// Mitsubishi GX Developer project: 12-202_20140305   PLC: FX3U

PROGRAM MAIN
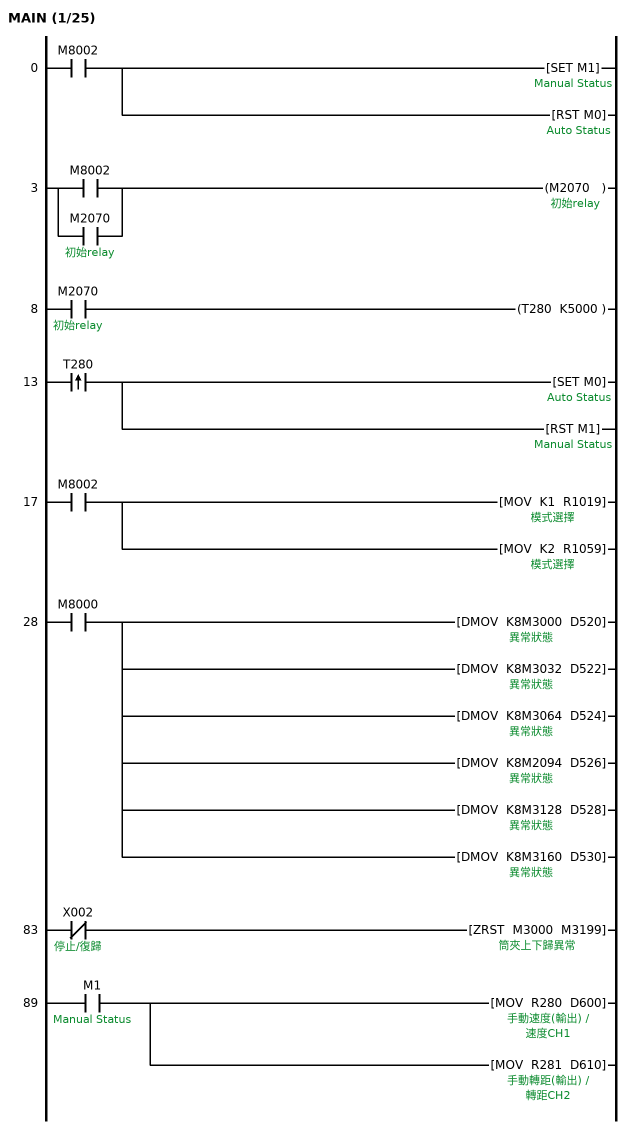
0     LD      M8002
      SET     M1  ; Manual Status
      RST     M0  ; Auto Status
3     LD      M8002
      OR      M2070  ; 初始relay
      OUT     M2070  ; 初始relay
8     LD      M2070  ; 初始relay
      OUT     T280 K5000
13    LDP     T280
      SET     M0  ; Auto Status
      RST     M1  ; Manual Status
17    LD      M8002
      MOV     K1 R1019  ; 模式選擇
      MOV     K2 R1059  ; 模式選擇
28    LD      M8000
      DMOV    K8M3000 D520  ; 筒夾上下歸異常 / 異常狀態
      DMOV    K8M3032 D522  ; 異常狀態
      DMOV    K8M3064 D524  ; 異常狀態
      DMOV    K8M2094 D526  ; 異常狀態
      DMOV    K8M3128 D528  ; 異常狀態
      DMOV    K8M3160 D530  ; 異常狀態
83    LDI     X002  ; 停止/復歸
      ZRST    M3000 M3199
89    LD      M1  ; Manual Status
      MOV     R280 D600  ; 手動速度(輸出) / 速度CH1
      MOV     R281 D610  ; 手動轉距(輸出) / 轉距CH2
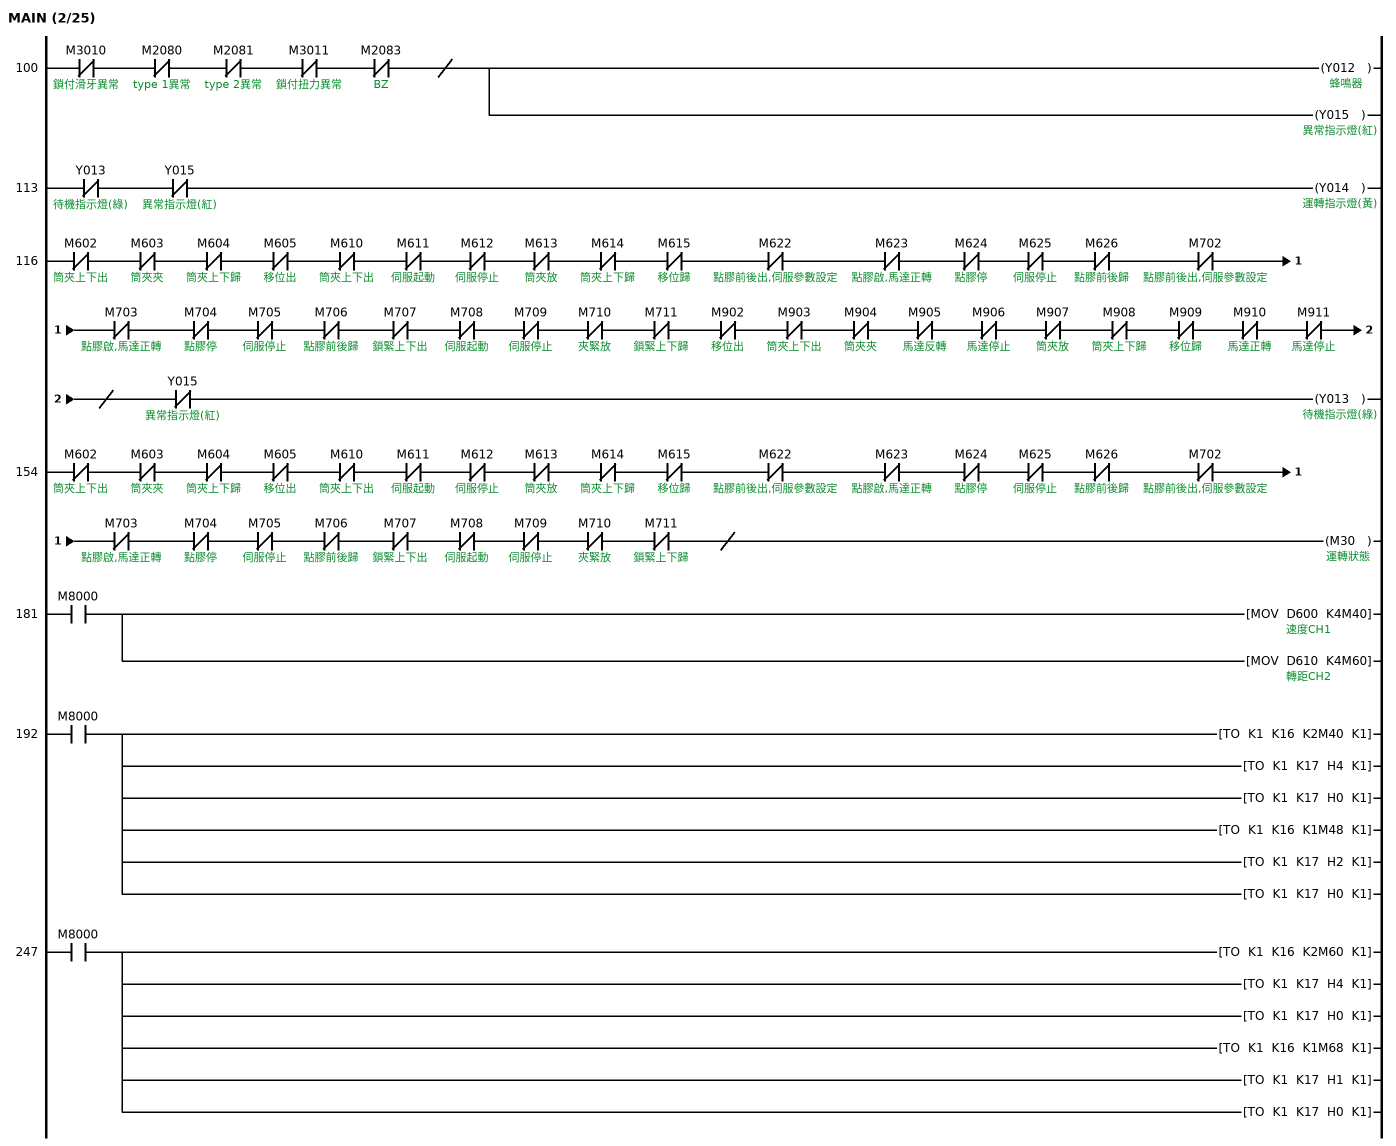
100   LDI     M3010  ; 鎖付滑牙異常
      ANI     M2080  ; type 1異常
      ANI     M2081  ; type 2異常
      ANI     M3011  ; 鎖付扭力異常
      ANI     M2083  ; BZ
      INV
      OUT     Y012  ; 蜂鳴器
      OUT     Y015  ; 異常指示燈(紅)
113   LDI     Y013  ; 待機指示燈(綠)
      ANI     Y015  ; 異常指示燈(紅)
      OUT     Y014  ; 運轉指示燈(黃)
116   LDI     M602  ; 筒夾上下出
      ANI     M603  ; 筒夾夾
      ANI     M604  ; 筒夾上下歸
      ANI     M605  ; 移位出
      ANI     M610  ; 筒夾上下出
      ANI     M611  ; 伺服起動
      ANI     M612  ; 伺服停止
      ANI     M613  ; 筒夾放
      ANI     M614  ; 筒夾上下歸
      ANI     M615  ; 移位歸
      ANI     M622  ; 點膠前後出,伺服參數設定
      ANI     M623  ; 點膠啟,馬達正轉
      ANI     M624  ; 點膠停
      ANI     M625  ; 伺服停止
      ANI     M626  ; 點膠前後歸
      ANI     M702  ; 點膠前後出,伺服參數設定
      ANI     M703  ; 點膠啟,馬達正轉
      ANI     M704  ; 點膠停
      ANI     M705  ; 伺服停止
      ANI     M706  ; 點膠前後歸
      ANI     M707  ; 鎖緊上下出
      ANI     M708  ; 伺服起動
      ANI     M709  ; 伺服停止
      ANI     M710  ; 夾緊放
      ANI     M711  ; 鎖緊上下歸
      ANI     M902  ; 移位出
      ANI     M903  ; 筒夾上下出
      ANI     M904  ; 筒夾夾
      ANI     M905  ; 馬達反轉
      ANI     M906  ; 馬達停止
      ANI     M907  ; 筒夾放
      ANI     M908  ; 筒夾上下歸
      ANI     M909  ; 移位歸
      ANI     M910  ; 馬達正轉
      ANI     M911  ; 馬達停止
      INV
      ANI     Y015  ; 異常指示燈(紅)
      OUT     Y013  ; 待機指示燈(綠)
154   LDI     M602  ; 筒夾上下出
      ANI     M603  ; 筒夾夾
      ANI     M604  ; 筒夾上下歸
      ANI     M605  ; 移位出
      ANI     M610  ; 筒夾上下出
      ANI     M611  ; 伺服起動
      ANI     M612  ; 伺服停止
      ANI     M613  ; 筒夾放
      ANI     M614  ; 筒夾上下歸
      ANI     M615  ; 移位歸
      ANI     M622  ; 點膠前後出,伺服參數設定
      ANI     M623  ; 點膠啟,馬達正轉
      ANI     M624  ; 點膠停
      ANI     M625  ; 伺服停止
      ANI     M626  ; 點膠前後歸
      ANI     M702  ; 點膠前後出,伺服參數設定
      ANI     M703  ; 點膠啟,馬達正轉
      ANI     M704  ; 點膠停
      ANI     M705  ; 伺服停止
      ANI     M706  ; 點膠前後歸
      ANI     M707  ; 鎖緊上下出
      ANI     M708  ; 伺服起動
      ANI     M709  ; 伺服停止
      ANI     M710  ; 夾緊放
      ANI     M711  ; 鎖緊上下歸
      INV
      OUT     M30  ; 運轉狀態
181   LD      M8000
      MOV     D600 K4M40  ; DA用
      MOV     D610 K4M60  ; DA用
192   LD      M8000
      TO      K1 K16 K2M40 K1
      TO      K1 K17 H4 K1
      TO      K1 K17 H0 K1
      TO      K1 K16 K1M48 K1  ; DA用
      TO      K1 K17 H2 K1
      TO      K1 K17 H0 K1
247   LD      M8000
      TO      K1 K16 K2M60 K1
      TO      K1 K17 H4 K1
      TO      K1 K17 H0 K1
      TO      K1 K16 K1M68 K1  ; DA用
      TO      K1 K17 H1 K1
      TO      K1 K17 H0 K1
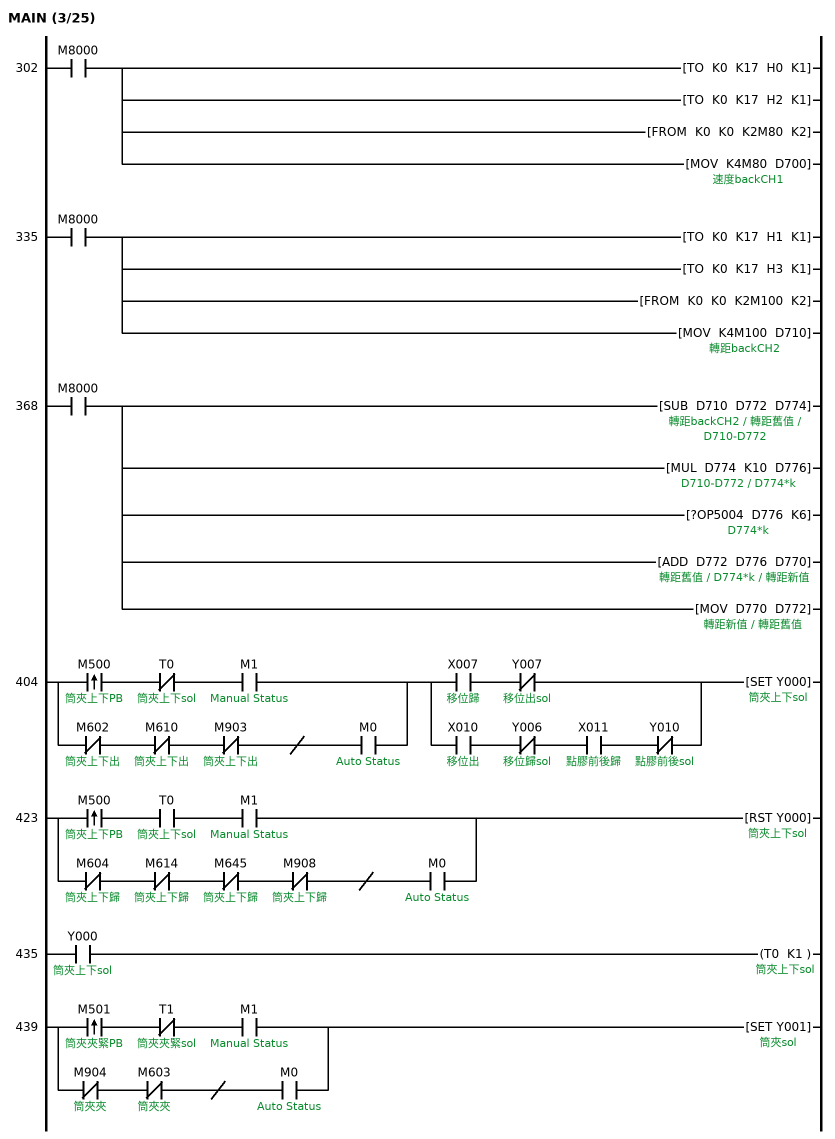
302   LD      M8000
      TO      K0 K17 H0 K1
      TO      K0 K17 H2 K1
      FROM    K0 K0 K2M80 K2  ; AD用
      MOV     K4M80 D700  ; 速度backCH1
335   LD      M8000
      TO      K0 K17 H1 K1
      TO      K0 K17 H3 K1
      FROM    K0 K0 K2M100 K2  ; AD用
      MOV     K4M100 D710  ; 轉距backCH2
368   LD      M8000
      SUB     D710 D772 D774  ; 轉距舊值 / D710-D772
      MUL     D774 K10 D776  ; D774*k
      ?OP5004 D776 K6
      ADD     D772 D776 D770  ; 轉距新值
      MOV     D770 D772
404   LDP     M500  ; 筒夾上下PB
      ANI     T0  ; 筒夾上下sol
      AND     M1  ; Manual Status
      LDI     M602  ; 筒夾上下出
      ANI     M610  ; 筒夾上下出
      ANI     M903  ; 筒夾上下出
      INV
      AND     M0  ; Auto Status
      ORB
      LD      X007  ; 移位歸
      ANI     Y007  ; 移位出sol
      LD      X010  ; 移位出
      ANI     Y006  ; 移位歸sol
      AND     X011  ; 點膠前後歸
      ANI     Y010  ; 點膠前後sol
      ORB
      ANB
      SET     Y000  ; 筒夾上下sol
423   LDP     M500  ; 筒夾上下PB
      AND     T0  ; 筒夾上下sol
      AND     M1  ; Manual Status
      LDI     M604  ; 筒夾上下歸
      ANI     M614  ; 筒夾上下歸
      ANI     M645  ; 筒夾上下歸
      ANI     M908  ; 筒夾上下歸
      INV
      AND     M0  ; Auto Status
      ORB
      RST     Y000  ; 筒夾上下sol
435   LD      Y000  ; 筒夾上下sol
      OUT     T0 K1  ; 筒夾上下sol
439   LDP     M501  ; 筒夾夾緊PB
      ANI     T1  ; 筒夾夾緊sol
      AND     M1  ; Manual Status
      LDI     M904  ; 筒夾夾
      ANI     M603  ; 筒夾夾
      INV
      AND     M0  ; Auto Status
      ORB
      SET     Y001  ; 筒夾sol
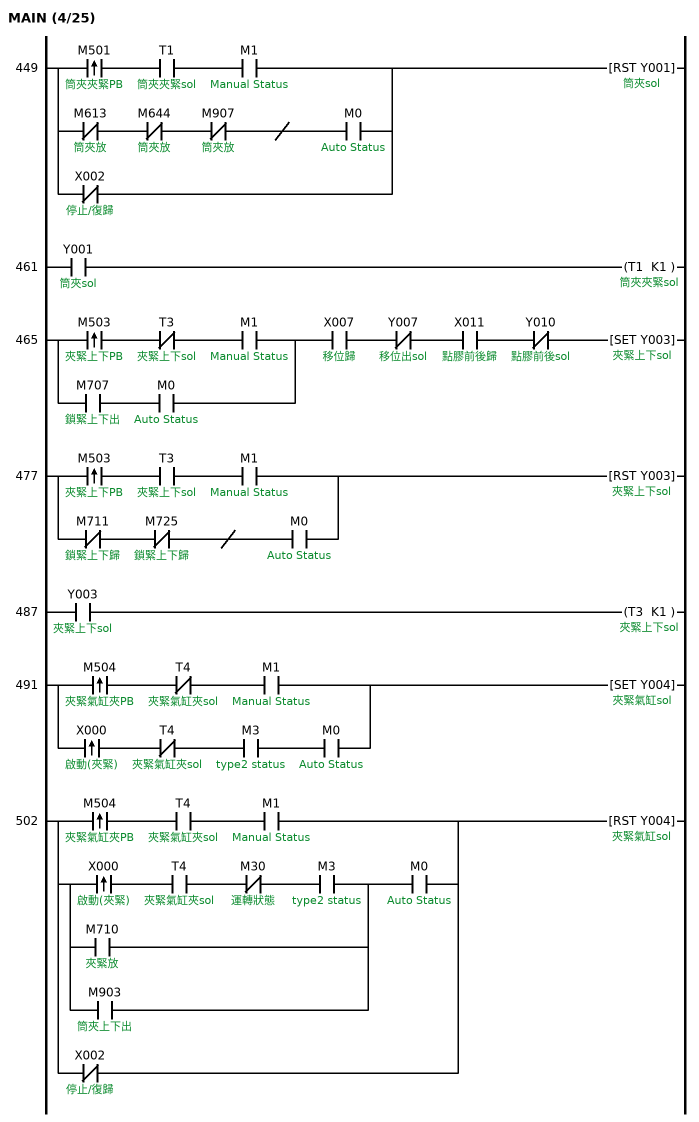
449   LDP     M501  ; 筒夾夾緊PB
      AND     T1  ; 筒夾夾緊sol
      AND     M1  ; Manual Status
      LDI     M613  ; 筒夾放
      ANI     M644  ; 筒夾放
      ANI     M907  ; 筒夾放
      INV
      AND     M0  ; Auto Status
      ORB
      ORI     X002  ; 停止/復歸
      RST     Y001  ; 筒夾sol
461   LD      Y001  ; 筒夾sol
      OUT     T1 K1  ; 筒夾夾緊sol
465   LDP     M503  ; 夾緊上下PB
      ANI     T3  ; 夾緊上下sol
      AND     M1  ; Manual Status
      LD      M707  ; 鎖緊上下出
      AND     M0  ; Auto Status
      ORB
      AND     X007  ; 移位歸
      ANI     Y007  ; 移位出sol
      AND     X011  ; 點膠前後歸
      ANI     Y010  ; 點膠前後sol
      SET     Y003  ; 夾緊上下sol
477   LDP     M503  ; 夾緊上下PB
      AND     T3  ; 夾緊上下sol
      AND     M1  ; Manual Status
      LDI     M711  ; 鎖緊上下歸
      ANI     M725  ; 鎖緊上下歸
      INV
      AND     M0  ; Auto Status
      ORB
      RST     Y003  ; 夾緊上下sol
487   LD      Y003  ; 夾緊上下sol
      OUT     T3 K1  ; 夾緊上下sol
491   LDP     M504  ; 夾緊氣缸夾PB
      ANI     T4  ; 夾緊氣缸夾sol
      AND     M1  ; Manual Status
      LDP     X000  ; 啟動(夾緊)
      ANI     T4  ; 夾緊氣缸夾sol
      AND     M3  ; type2 status
      AND     M0  ; Auto Status
      ORB
      SET     Y004  ; 夾緊氣缸sol
502   LDP     M504  ; 夾緊氣缸夾PB
      AND     T4  ; 夾緊氣缸夾sol
      AND     M1  ; Manual Status
      LDP     X000  ; 啟動(夾緊)
      AND     T4  ; 夾緊氣缸夾sol
      ANI     M30  ; 運轉狀態
      AND     M3  ; type2 status
      OR      M710  ; 夾緊放
      OR      M903  ; 筒夾上下出
      AND     M0  ; Auto Status
      ORB
      ORI     X002  ; 停止/復歸
      RST     Y004  ; 夾緊氣缸sol
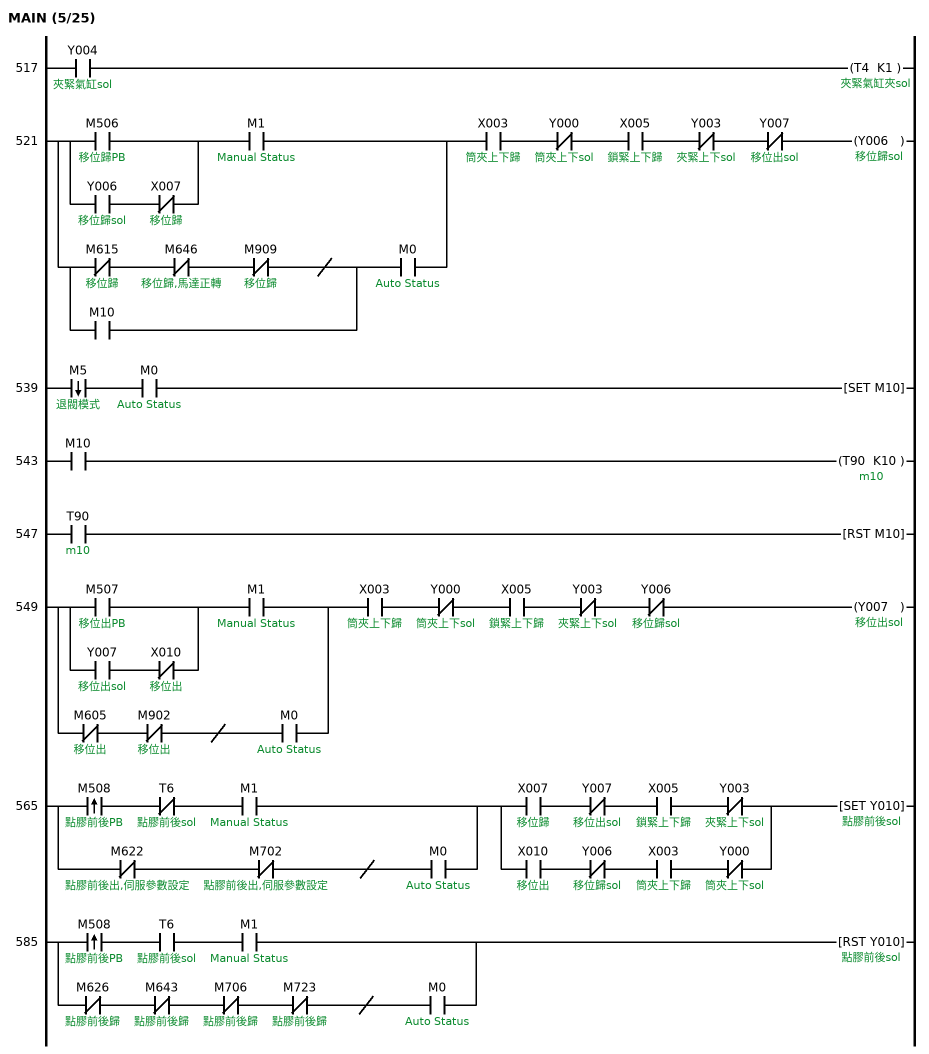
517   LD      Y004  ; 夾緊氣缸sol
      OUT     T4 K1  ; 夾緊氣缸夾sol
521   LD      M506  ; 移位歸PB
      LD      Y006  ; 移位歸sol
      ANI     X007  ; 移位歸
      ORB
      AND     M1  ; Manual Status
      LDI     M615  ; 移位歸
      ANI     M646  ; 移位歸,馬達正轉
      ANI     M909  ; 移位歸
      INV
      OR      M10
      AND     M0  ; Auto Status
      ORB
      AND     X003  ; 筒夾上下歸
      ANI     Y000  ; 筒夾上下sol
      AND     X005  ; 鎖緊上下歸
      ANI     Y003  ; 夾緊上下sol
      ANI     Y007  ; 移位出sol
      OUT     Y006  ; 移位歸sol
539   LDF     M5  ; 退閥模式
      AND     M0  ; Auto Status
      SET     M10
543   LD      M10
      OUT     T90 K10  ; m10
547   LD      T90  ; m10
      RST     M10
549   LD      M507  ; 移位出PB
      LD      Y007  ; 移位出sol
      ANI     X010  ; 移位出
      ORB
      AND     M1  ; Manual Status
      LDI     M605  ; 移位出
      ANI     M902  ; 移位出
      INV
      AND     M0  ; Auto Status
      ORB
      AND     X003  ; 筒夾上下歸
      ANI     Y000  ; 筒夾上下sol
      AND     X005  ; 鎖緊上下歸
      ANI     Y003  ; 夾緊上下sol
      ANI     Y006  ; 移位歸sol
      OUT     Y007  ; 移位出sol
565   LDP     M508  ; 點膠前後PB
      ANI     T6  ; 點膠前後sol
      AND     M1  ; Manual Status
      LDI     M622  ; 點膠前後出,伺服參數設定
      ANI     M702  ; 點膠前後出,伺服參數設定
      INV
      AND     M0  ; Auto Status
      ORB
      LD      X007  ; 移位歸
      ANI     Y007  ; 移位出sol
      AND     X005  ; 鎖緊上下歸
      ANI     Y003  ; 夾緊上下sol
      LD      X010  ; 移位出
      ANI     Y006  ; 移位歸sol
      AND     X003  ; 筒夾上下歸
      ANI     Y000  ; 筒夾上下sol
      ORB
      ANB
      SET     Y010  ; 點膠前後sol
585   LDP     M508  ; 點膠前後PB
      AND     T6  ; 點膠前後sol
      AND     M1  ; Manual Status
      LDI     M626  ; 點膠前後歸
      ANI     M643  ; 點膠前後歸
      ANI     M706  ; 點膠前後歸
      ANI     M723  ; 點膠前後歸
      INV
      AND     M0  ; Auto Status
      ORB
      RST     Y010  ; 點膠前後sol
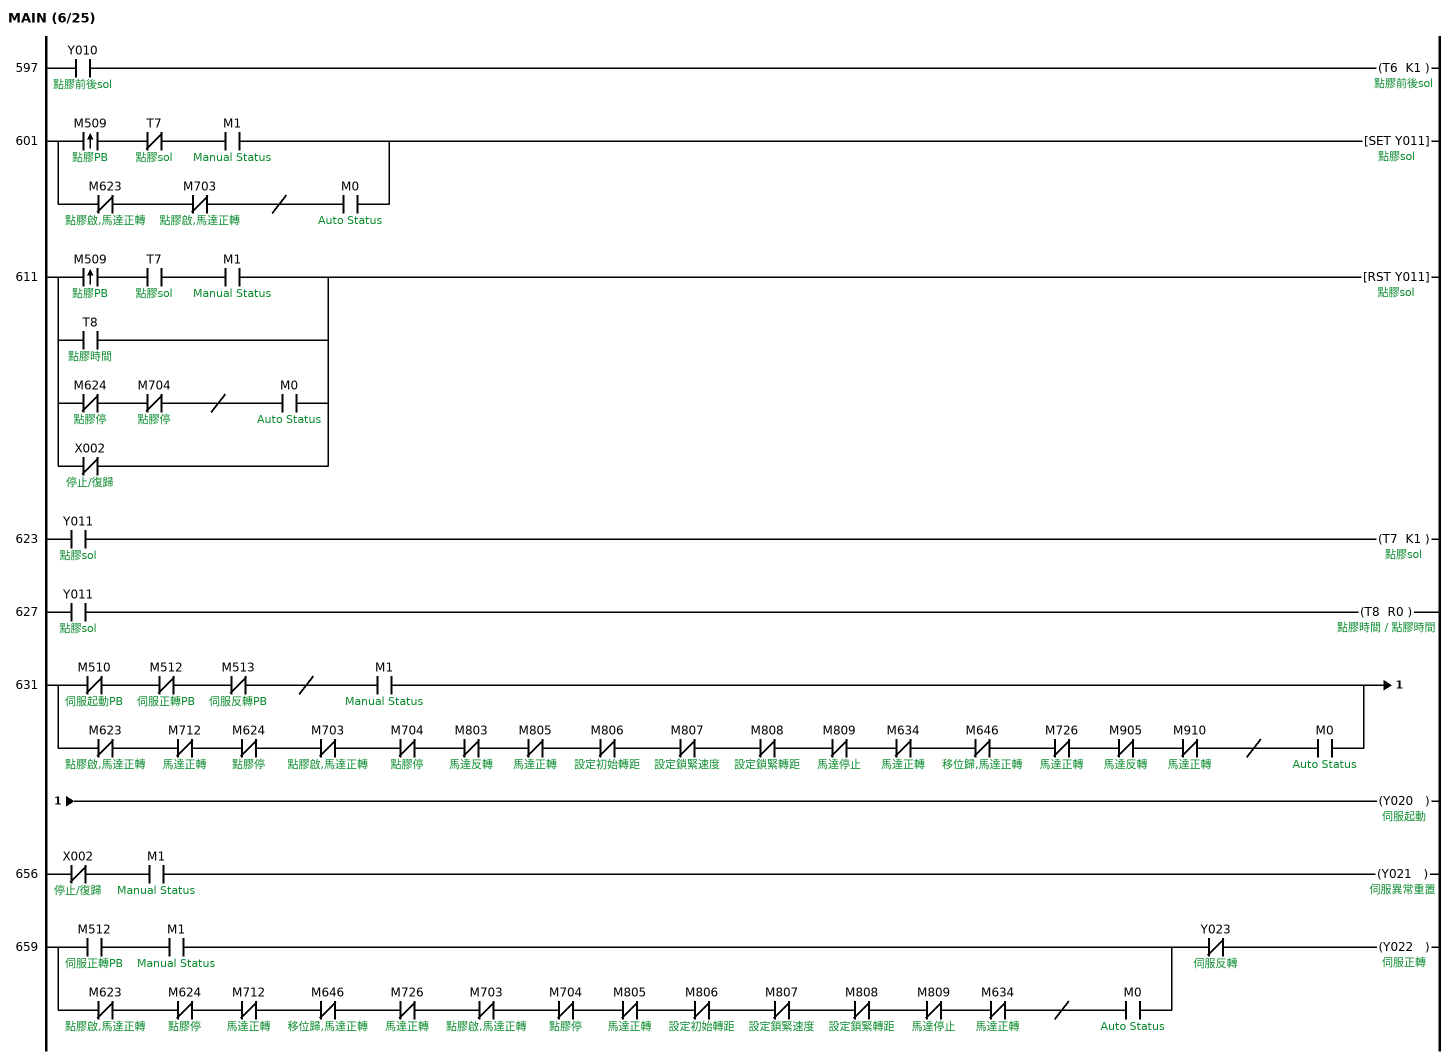
597   LD      Y010  ; 點膠前後sol
      OUT     T6 K1  ; 點膠前後sol
601   LDP     M509  ; 點膠PB
      ANI     T7  ; 點膠sol
      AND     M1  ; Manual Status
      LDI     M623  ; 點膠啟,馬達正轉
      ANI     M703  ; 點膠啟,馬達正轉
      INV
      AND     M0  ; Auto Status
      ORB
      SET     Y011  ; 點膠sol
611   LDP     M509  ; 點膠PB
      AND     T7  ; 點膠sol
      AND     M1  ; Manual Status
      OR      T8  ; 點膠時間
      LDI     M624  ; 點膠停
      ANI     M704  ; 點膠停
      INV
      AND     M0  ; Auto Status
      ORB
      ORI     X002  ; 停止/復歸
      RST     Y011  ; 點膠sol
623   LD      Y011  ; 點膠sol
      OUT     T7 K1  ; 點膠sol
627   LD      Y011  ; 點膠sol
      OUT     T8 R0  ; 點膠時間 / 點膠時間
631   LDI     M510  ; 伺服起動PB
      ANI     M512  ; 伺服正轉PB
      ANI     M513  ; 伺服反轉PB
      INV
      AND     M1  ; Manual Status
      LDI     M623  ; 點膠啟,馬達正轉
      ANI     M712  ; 馬達正轉
      ANI     M624  ; 點膠停
      ANI     M703  ; 點膠啟,馬達正轉
      ANI     M704  ; 點膠停
      ANI     M803  ; 馬達反轉
      ANI     M805  ; 馬達正轉
      ANI     M806  ; 設定初始轉距
      ANI     M807  ; 設定鎖緊速度
      ANI     M808  ; 設定鎖緊轉距
      ANI     M809  ; 馬達停止
      ANI     M634  ; 馬達正轉
      ANI     M646  ; 移位歸,馬達正轉
      ANI     M726  ; 馬達正轉
      ANI     M905  ; 馬達反轉
      ANI     M910  ; 馬達正轉
      INV
      AND     M0  ; Auto Status
      ORB
      OUT     Y020  ; 伺服起動
656   LDI     X002  ; 停止/復歸
      AND     M1  ; Manual Status
      OUT     Y021  ; 伺服異常重置
659   LD      M512  ; 伺服正轉PB
      AND     M1  ; Manual Status
      LDI     M623  ; 點膠啟,馬達正轉
      ANI     M624  ; 點膠停
      ANI     M712  ; 馬達正轉
      ANI     M646  ; 移位歸,馬達正轉
      ANI     M726  ; 馬達正轉
      ANI     M703  ; 點膠啟,馬達正轉
      ANI     M704  ; 點膠停
      ANI     M805  ; 馬達正轉
      ANI     M806  ; 設定初始轉距
      ANI     M807  ; 設定鎖緊速度
      ANI     M808  ; 設定鎖緊轉距
      ANI     M809  ; 馬達停止
      ANI     M634  ; 馬達正轉
      INV
      AND     M0  ; Auto Status
      ORB
      ANI     Y023  ; 伺服反轉
      OUT     Y022  ; 伺服正轉
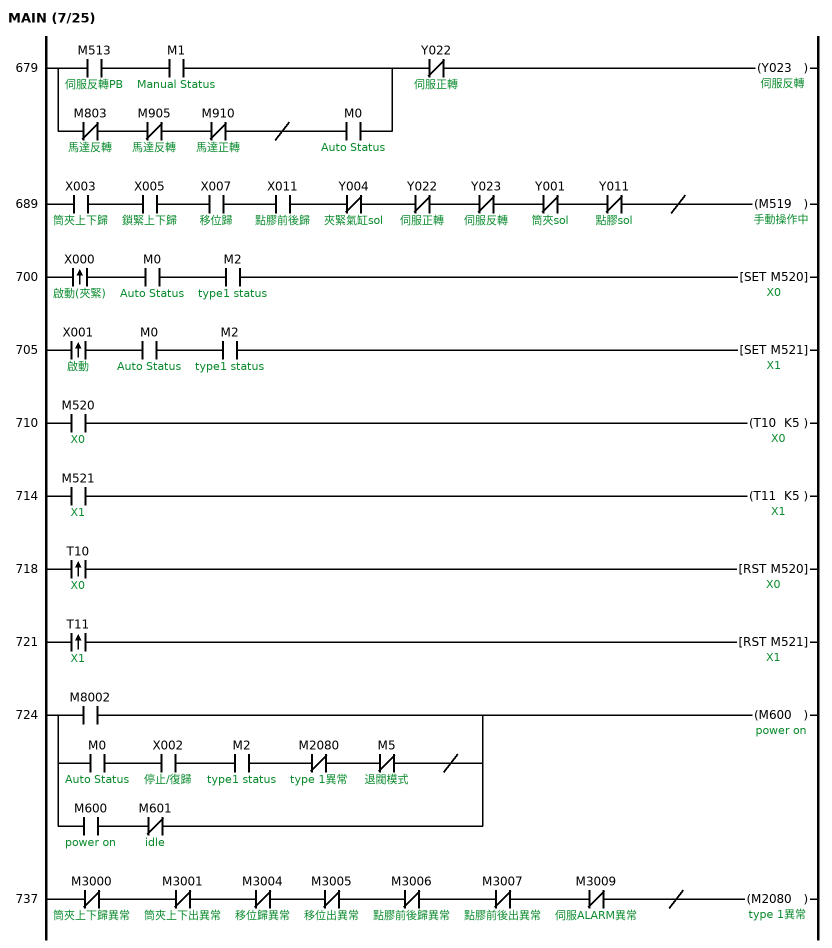
679   LD      M513  ; 伺服反轉PB
      AND     M1  ; Manual Status
      LDI     M803  ; 馬達反轉
      ANI     M905  ; 馬達反轉
      ANI     M910  ; 馬達正轉
      INV
      AND     M0  ; Auto Status
      ORB
      ANI     Y022  ; 伺服正轉
      OUT     Y023  ; 伺服反轉
689   LD      X003  ; 筒夾上下歸
      AND     X005  ; 鎖緊上下歸
      AND     X007  ; 移位歸
      AND     X011  ; 點膠前後歸
      ANI     Y004  ; 夾緊氣缸sol
      ANI     Y022  ; 伺服正轉
      ANI     Y023  ; 伺服反轉
      ANI     Y001  ; 筒夾sol
      ANI     Y011  ; 點膠sol
      INV
      OUT     M519  ; 手動操作中
700   LDP     X000  ; 啟動(夾緊)
      AND     M0  ; Auto Status
      AND     M2  ; type1 status
      SET     M520  ; X0
705   LDP     X001  ; 啟動
      AND     M0  ; Auto Status
      AND     M2  ; type1 status
      SET     M521  ; X1
710   LD      M520  ; X0
      OUT     T10 K5  ; X0
714   LD      M521  ; X1
      OUT     T11 K5  ; X1
718   LDP     T10  ; X0
      RST     M520  ; X0
721   LDP     T11  ; X1
      RST     M521  ; X1
724   LD      M8002
      LD      M0  ; Auto Status
      AND     X002  ; 停止/復歸
      AND     M2  ; type1 status
      ANI     M2080  ; type 1異常
      ANI     M5  ; 退閥模式
      INV
      ORB
      LD      M600  ; power on
      ANI     M601  ; idle
      ORB
      OUT     M600  ; power on
737   LDI     M3000  ; 筒夾上下歸異常
      ANI     M3001  ; 筒夾上下出異常
      ANI     M3004  ; 移位歸異常
      ANI     M3005  ; 移位出異常
      ANI     M3006  ; 點膠前後歸異常
      ANI     M3007  ; 點膠前後出異常
      ANI     M3009  ; 伺服ALARM異常
      INV
      OUT     M2080  ; type 1異常
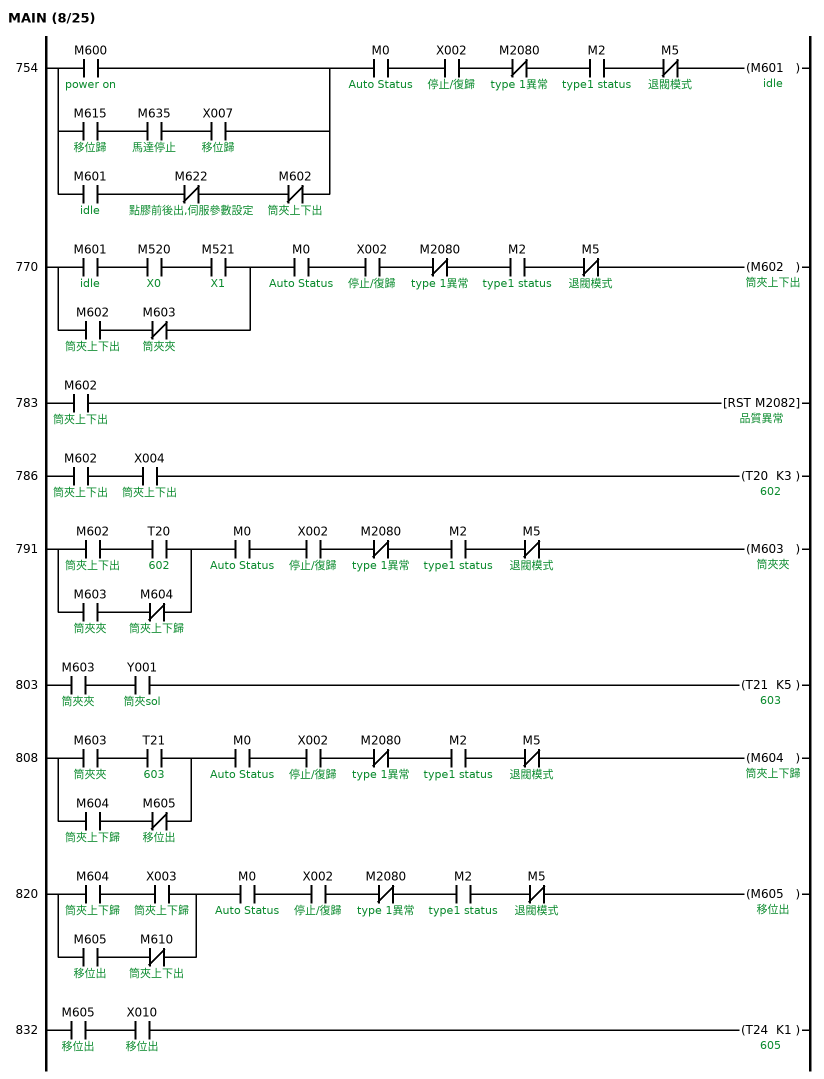
754   LD      M600  ; power on
      LD      M615  ; 移位歸
      AND     M635  ; 馬達停止
      AND     X007  ; 移位歸
      ORB
      LD      M601  ; idle
      ANI     M622  ; 點膠前後出,伺服參數設定
      ANI     M602  ; 筒夾上下出
      ORB
      AND     M0  ; Auto Status
      AND     X002  ; 停止/復歸
      ANI     M2080  ; type 1異常
      AND     M2  ; type1 status
      ANI     M5  ; 退閥模式
      OUT     M601  ; idle
770   LD      M601  ; idle
      AND     M520  ; X0
      AND     M521  ; X1
      LD      M602  ; 筒夾上下出
      ANI     M603  ; 筒夾夾
      ORB
      AND     M0  ; Auto Status
      AND     X002  ; 停止/復歸
      ANI     M2080  ; type 1異常
      AND     M2  ; type1 status
      ANI     M5  ; 退閥模式
      OUT     M602  ; 筒夾上下出
783   LD      M602  ; 筒夾上下出
      RST     M2082  ; 品質異常
786   LD      M602  ; 筒夾上下出
      AND     X004  ; 筒夾上下出
      OUT     T20 K3  ; 602
791   LD      M602  ; 筒夾上下出
      AND     T20  ; 602
      LD      M603  ; 筒夾夾
      ANI     M604  ; 筒夾上下歸
      ORB
      AND     M0  ; Auto Status
      AND     X002  ; 停止/復歸
      ANI     M2080  ; type 1異常
      AND     M2  ; type1 status
      ANI     M5  ; 退閥模式
      OUT     M603  ; 筒夾夾
803   LD      M603  ; 筒夾夾
      AND     Y001  ; 筒夾sol
      OUT     T21 K5  ; 603
808   LD      M603  ; 筒夾夾
      AND     T21  ; 603
      LD      M604  ; 筒夾上下歸
      ANI     M605  ; 移位出
      ORB
      AND     M0  ; Auto Status
      AND     X002  ; 停止/復歸
      ANI     M2080  ; type 1異常
      AND     M2  ; type1 status
      ANI     M5  ; 退閥模式
      OUT     M604  ; 筒夾上下歸
820   LD      M604  ; 筒夾上下歸
      AND     X003  ; 筒夾上下歸
      LD      M605  ; 移位出
      ANI     M610  ; 筒夾上下出
      ORB
      AND     M0  ; Auto Status
      AND     X002  ; 停止/復歸
      ANI     M2080  ; type 1異常
      AND     M2  ; type1 status
      ANI     M5  ; 退閥模式
      OUT     M605  ; 移位出
832   LD      M605  ; 移位出
      AND     X010  ; 移位出
      OUT     T24 K1  ; 605
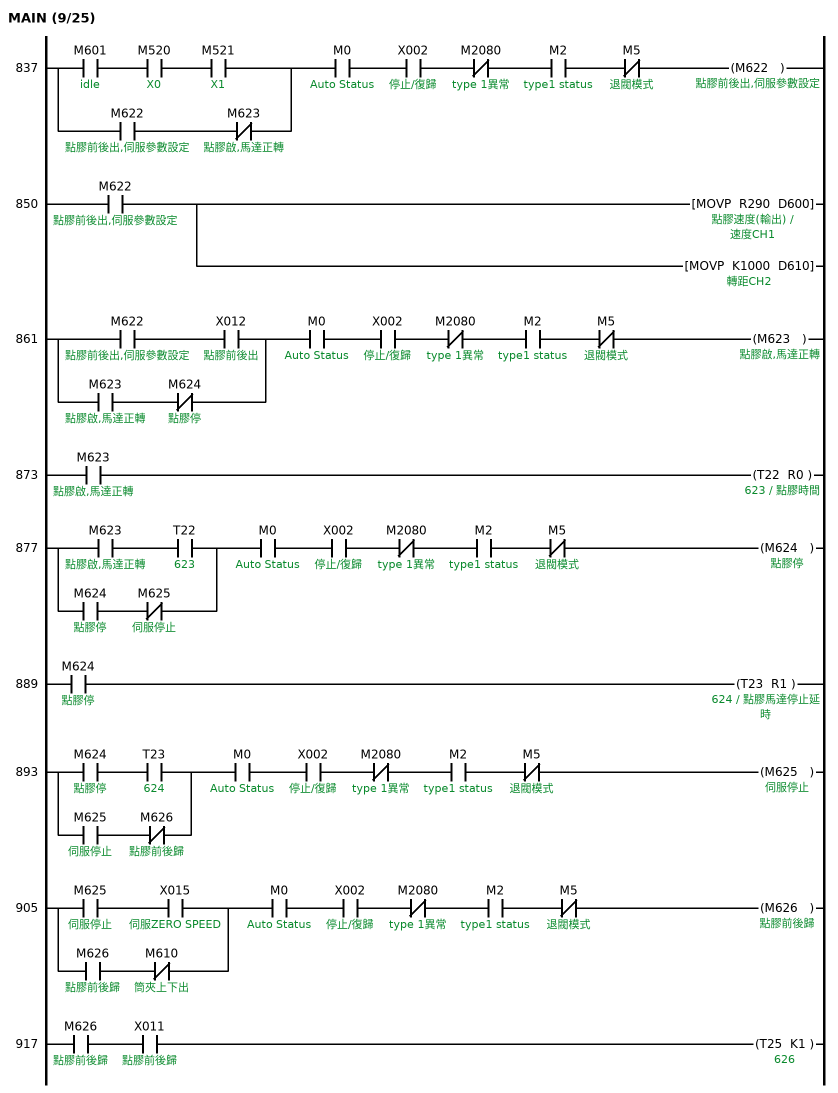
837   LD      M601  ; idle
      AND     M520  ; X0
      AND     M521  ; X1
      LD      M622  ; 點膠前後出,伺服參數設定
      ANI     M623  ; 點膠啟,馬達正轉
      ORB
      AND     M0  ; Auto Status
      AND     X002  ; 停止/復歸
      ANI     M2080  ; type 1異常
      AND     M2  ; type1 status
      ANI     M5  ; 退閥模式
      OUT     M622  ; 點膠前後出,伺服參數設定
850   LD      M622  ; 點膠前後出,伺服參數設定
      MOVP    R290 D600  ; 點膠速度(輸出)
      MOVP    K1000 D610
861   LD      M622  ; 點膠前後出,伺服參數設定
      AND     X012  ; 點膠前後出
      LD      M623  ; 點膠啟,馬達正轉
      ANI     M624  ; 點膠停
      ORB
      AND     M0  ; Auto Status
      AND     X002  ; 停止/復歸
      ANI     M2080  ; type 1異常
      AND     M2  ; type1 status
      ANI     M5  ; 退閥模式
      OUT     M623  ; 點膠啟,馬達正轉
873   LD      M623  ; 點膠啟,馬達正轉
      OUT     T22 R0  ; 623 / 點膠時間
877   LD      M623  ; 點膠啟,馬達正轉
      AND     T22  ; 623
      LD      M624  ; 點膠停
      ANI     M625  ; 伺服停止
      ORB
      AND     M0  ; Auto Status
      AND     X002  ; 停止/復歸
      ANI     M2080  ; type 1異常
      AND     M2  ; type1 status
      ANI     M5  ; 退閥模式
      OUT     M624  ; 點膠停
889   LD      M624  ; 點膠停
      OUT     T23 R1  ; 624 / 點膠馬達停止延時
893   LD      M624  ; 點膠停
      AND     T23  ; 624
      LD      M625  ; 伺服停止
      ANI     M626  ; 點膠前後歸
      ORB
      AND     M0  ; Auto Status
      AND     X002  ; 停止/復歸
      ANI     M2080  ; type 1異常
      AND     M2  ; type1 status
      ANI     M5  ; 退閥模式
      OUT     M625  ; 伺服停止
905   LD      M625  ; 伺服停止
      AND     X015  ; 伺服ZERO SPEED
      LD      M626  ; 點膠前後歸
      ANI     M610  ; 筒夾上下出
      ORB
      AND     M0  ; Auto Status
      AND     X002  ; 停止/復歸
      ANI     M2080  ; type 1異常
      AND     M2  ; type1 status
      ANI     M5  ; 退閥模式
      OUT     M626  ; 點膠前後歸
917   LD      M626  ; 點膠前後歸
      AND     X011  ; 點膠前後歸
      OUT     T25 K1  ; 626
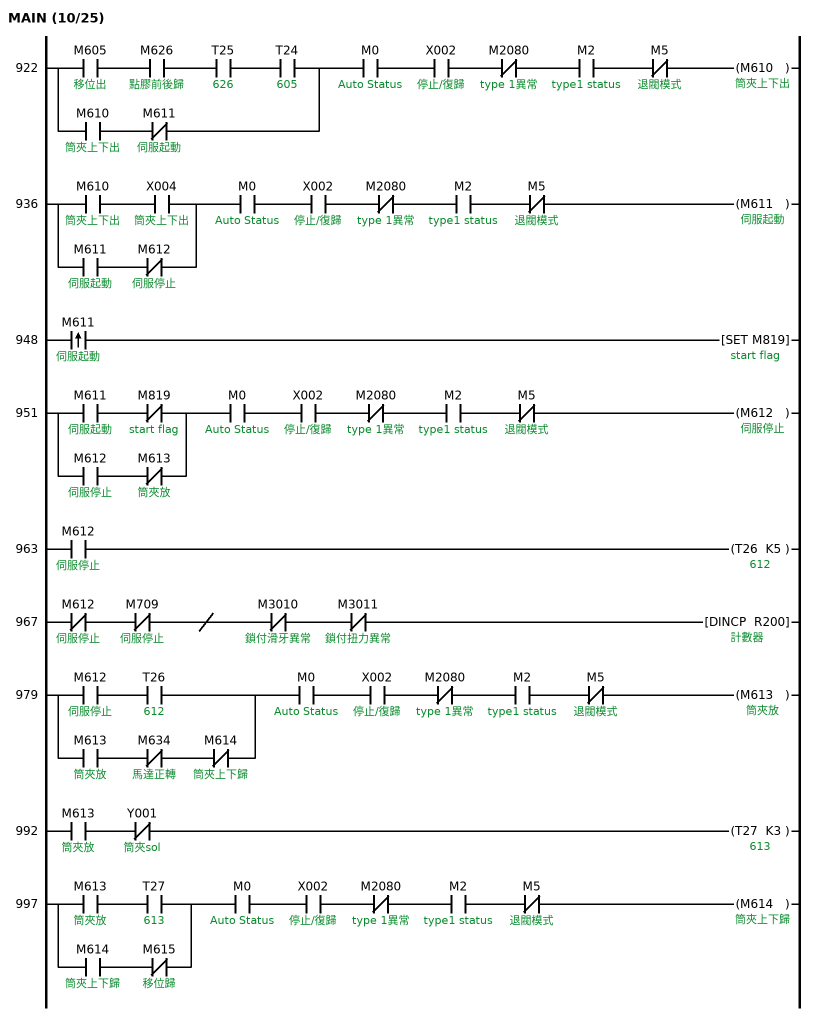
922   LD      M605  ; 移位出
      AND     M626  ; 點膠前後歸
      AND     T25  ; 626
      AND     T24  ; 605
      LD      M610  ; 筒夾上下出
      ANI     M611  ; 伺服起動
      ORB
      AND     M0  ; Auto Status
      AND     X002  ; 停止/復歸
      ANI     M2080  ; type 1異常
      AND     M2  ; type1 status
      ANI     M5  ; 退閥模式
      OUT     M610  ; 筒夾上下出
936   LD      M610  ; 筒夾上下出
      AND     X004  ; 筒夾上下出
      LD      M611  ; 伺服起動
      ANI     M612  ; 伺服停止
      ORB
      AND     M0  ; Auto Status
      AND     X002  ; 停止/復歸
      ANI     M2080  ; type 1異常
      AND     M2  ; type1 status
      ANI     M5  ; 退閥模式
      OUT     M611  ; 伺服起動
948   LDP     M611  ; 伺服起動
      SET     M819  ; start flag
951   LD      M611  ; 伺服起動
      ANI     M819  ; start flag
      LD      M612  ; 伺服停止
      ANI     M613  ; 筒夾放
      ORB
      AND     M0  ; Auto Status
      AND     X002  ; 停止/復歸
      ANI     M2080  ; type 1異常
      AND     M2  ; type1 status
      ANI     M5  ; 退閥模式
      OUT     M612  ; 伺服停止
963   LD      M612  ; 伺服停止
      OUT     T26 K5  ; 612
967   LDI     M612  ; 伺服停止
      ANI     M709  ; 伺服停止
      INV
      ANI     M3010  ; 鎖付滑牙異常
      ANI     M3011  ; 鎖付扭力異常
      DINCP   R200  ; 計數器
979   LD      M612  ; 伺服停止
      AND     T26  ; 612
      LD      M613  ; 筒夾放
      ANI     M634  ; 馬達正轉
      ANI     M614  ; 筒夾上下歸
      ORB
      AND     M0  ; Auto Status
      AND     X002  ; 停止/復歸
      ANI     M2080  ; type 1異常
      AND     M2  ; type1 status
      ANI     M5  ; 退閥模式
      OUT     M613  ; 筒夾放
992   LD      M613  ; 筒夾放
      ANI     Y001  ; 筒夾sol
      OUT     T27 K3  ; 613
997   LD      M613  ; 筒夾放
      AND     T27  ; 613
      LD      M614  ; 筒夾上下歸
      ANI     M615  ; 移位歸
      ORB
      AND     M0  ; Auto Status
      AND     X002  ; 停止/復歸
      ANI     M2080  ; type 1異常
      AND     M2  ; type1 status
      ANI     M5  ; 退閥模式
      OUT     M614  ; 筒夾上下歸
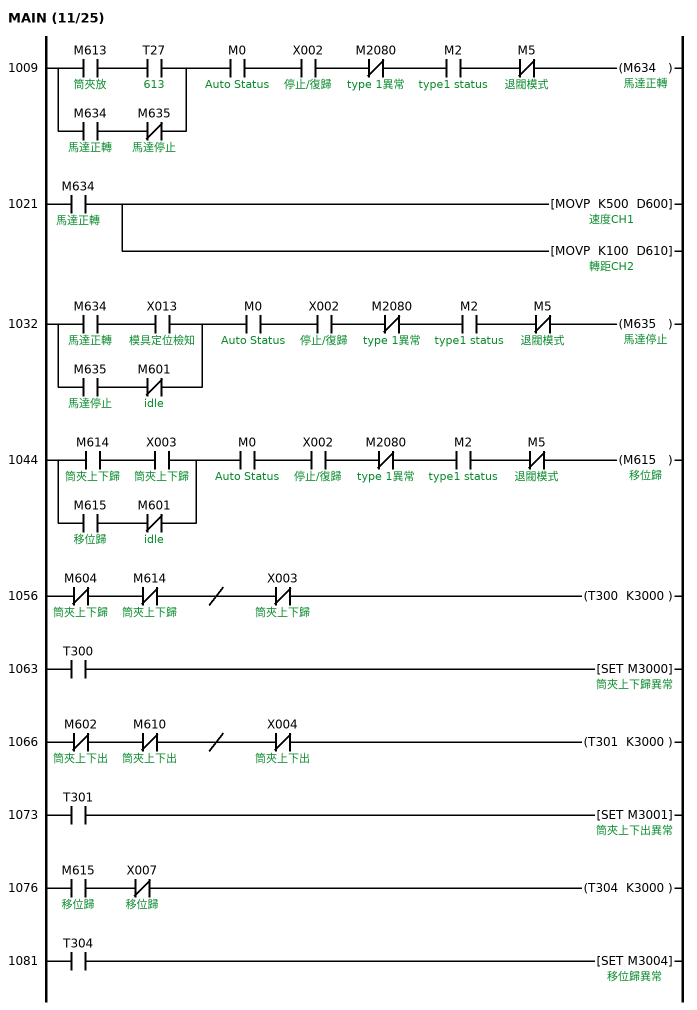
1009  LD      M613  ; 筒夾放
      AND     T27  ; 613
      LD      M634  ; 馬達正轉
      ANI     M635  ; 馬達停止
      ORB
      AND     M0  ; Auto Status
      AND     X002  ; 停止/復歸
      ANI     M2080  ; type 1異常
      AND     M2  ; type1 status
      ANI     M5  ; 退閥模式
      OUT     M634  ; 馬達正轉
1021  LD      M634  ; 馬達正轉
      MOVP    K500 D600
      MOVP    K100 D610
1032  LD      M634  ; 馬達正轉
      AND     X013  ; 模具定位檢知
      LD      M635  ; 馬達停止
      ANI     M601  ; idle
      ORB
      AND     M0  ; Auto Status
      AND     X002  ; 停止/復歸
      ANI     M2080  ; type 1異常
      AND     M2  ; type1 status
      ANI     M5  ; 退閥模式
      OUT     M635  ; 馬達停止
1044  LD      M614  ; 筒夾上下歸
      AND     X003  ; 筒夾上下歸
      LD      M615  ; 移位歸
      ANI     M601  ; idle
      ORB
      AND     M0  ; Auto Status
      AND     X002  ; 停止/復歸
      ANI     M2080  ; type 1異常
      AND     M2  ; type1 status
      ANI     M5  ; 退閥模式
      OUT     M615  ; 移位歸
1056  LDI     M604  ; 筒夾上下歸
      ANI     M614  ; 筒夾上下歸
      INV
      ANI     X003  ; 筒夾上下歸
      OUT     T300 K3000
1063  LD      T300
      SET     M3000  ; 筒夾上下歸異常
1066  LDI     M602  ; 筒夾上下出
      ANI     M610  ; 筒夾上下出
      INV
      ANI     X004  ; 筒夾上下出
      OUT     T301 K3000
1073  LD      T301
      SET     M3001  ; 筒夾上下出異常
1076  LD      M615  ; 移位歸
      ANI     X007  ; 移位歸
      OUT     T304 K3000
1081  LD      T304
      SET     M3004  ; 移位歸異常
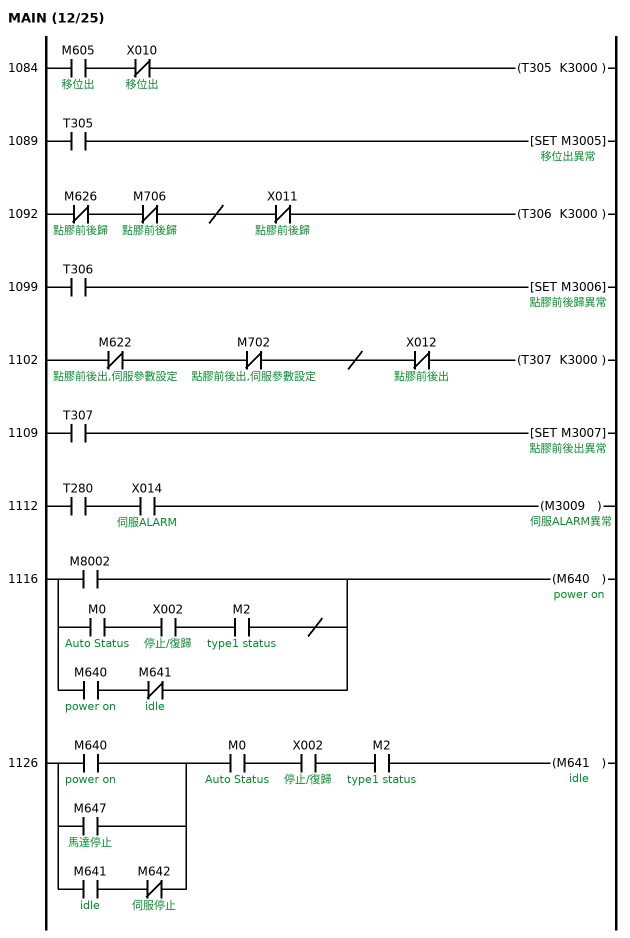
1084  LD      M605  ; 移位出
      ANI     X010  ; 移位出
      OUT     T305 K3000
1089  LD      T305
      SET     M3005  ; 移位出異常
1092  LDI     M626  ; 點膠前後歸
      ANI     M706  ; 點膠前後歸
      INV
      ANI     X011  ; 點膠前後歸
      OUT     T306 K3000
1099  LD      T306
      SET     M3006  ; 點膠前後歸異常
1102  LDI     M622  ; 點膠前後出,伺服參數設定
      ANI     M702  ; 點膠前後出,伺服參數設定
      INV
      ANI     X012  ; 點膠前後出
      OUT     T307 K3000
1109  LD      T307
      SET     M3007  ; 點膠前後出異常
1112  LD      T280
      AND     X014  ; 伺服ALARM
      OUT     M3009  ; 伺服ALARM異常
1116  LD      M8002
      LD      M0  ; Auto Status
      AND     X002  ; 停止/復歸
      AND     M2  ; type1 status
      INV
      ORB
      LD      M640  ; power on
      ANI     M641  ; idle
      ORB
      OUT     M640  ; power on
1126  LD      M640  ; power on
      OR      M647  ; 馬達停止
      LD      M641  ; idle
      ANI     M642  ; 伺服停止
      ORB
      AND     M0  ; Auto Status
      AND     X002  ; 停止/復歸
      AND     M2  ; type1 status
      OUT     M641  ; idle
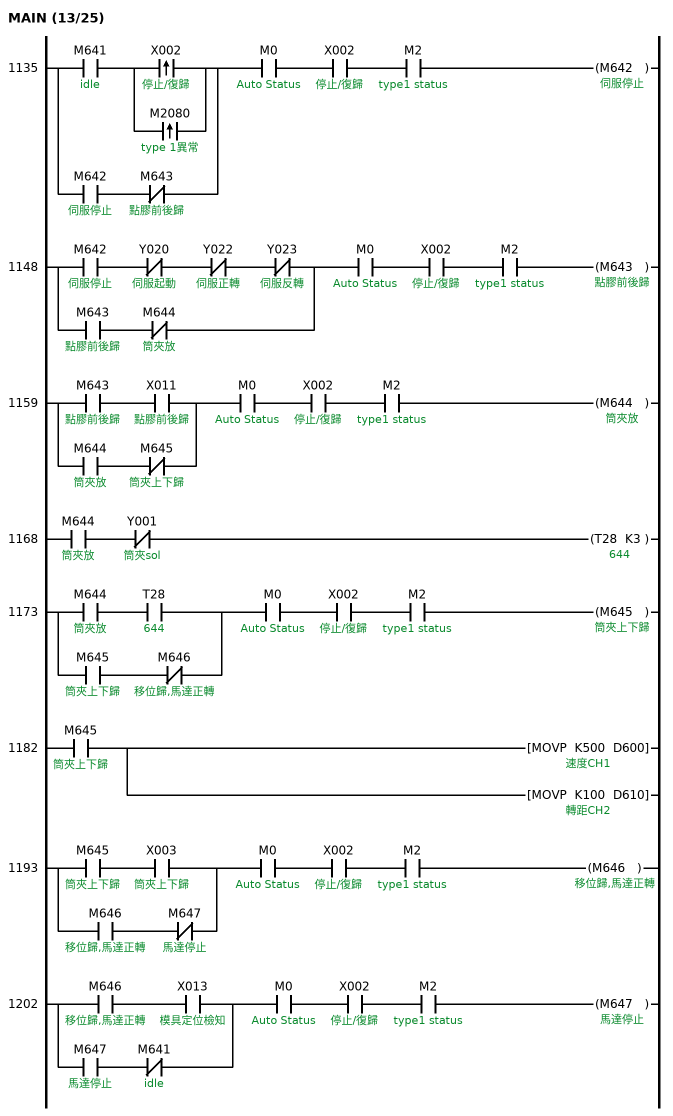
1135  LD      M641  ; idle
      LDP     X002  ; 停止/復歸
      ORP     M2080  ; type 1異常
      ANB
      LD      M642  ; 伺服停止
      ANI     M643  ; 點膠前後歸
      ORB
      AND     M0  ; Auto Status
      AND     X002  ; 停止/復歸
      AND     M2  ; type1 status
      OUT     M642  ; 伺服停止
1148  LD      M642  ; 伺服停止
      ANI     Y020  ; 伺服起動
      ANI     Y022  ; 伺服正轉
      ANI     Y023  ; 伺服反轉
      LD      M643  ; 點膠前後歸
      ANI     M644  ; 筒夾放
      ORB
      AND     M0  ; Auto Status
      AND     X002  ; 停止/復歸
      AND     M2  ; type1 status
      OUT     M643  ; 點膠前後歸
1159  LD      M643  ; 點膠前後歸
      AND     X011  ; 點膠前後歸
      LD      M644  ; 筒夾放
      ANI     M645  ; 筒夾上下歸
      ORB
      AND     M0  ; Auto Status
      AND     X002  ; 停止/復歸
      AND     M2  ; type1 status
      OUT     M644  ; 筒夾放
1168  LD      M644  ; 筒夾放
      ANI     Y001  ; 筒夾sol
      OUT     T28 K3  ; 644
1173  LD      M644  ; 筒夾放
      AND     T28  ; 644
      LD      M645  ; 筒夾上下歸
      ANI     M646  ; 移位歸,馬達正轉
      ORB
      AND     M0  ; Auto Status
      AND     X002  ; 停止/復歸
      AND     M2  ; type1 status
      OUT     M645  ; 筒夾上下歸
1182  LD      M645  ; 筒夾上下歸
      MOVP    K500 D600
      MOVP    K100 D610
1193  LD      M645  ; 筒夾上下歸
      AND     X003  ; 筒夾上下歸
      LD      M646  ; 移位歸,馬達正轉
      ANI     M647  ; 馬達停止
      ORB
      AND     M0  ; Auto Status
      AND     X002  ; 停止/復歸
      AND     M2  ; type1 status
      OUT     M646  ; 移位歸,馬達正轉
1202  LD      M646  ; 移位歸,馬達正轉
      AND     X013  ; 模具定位檢知
      LD      M647  ; 馬達停止
      ANI     M641  ; idle
      ORB
      AND     M0  ; Auto Status
      AND     X002  ; 停止/復歸
      AND     M2  ; type1 status
      OUT     M647  ; 馬達停止
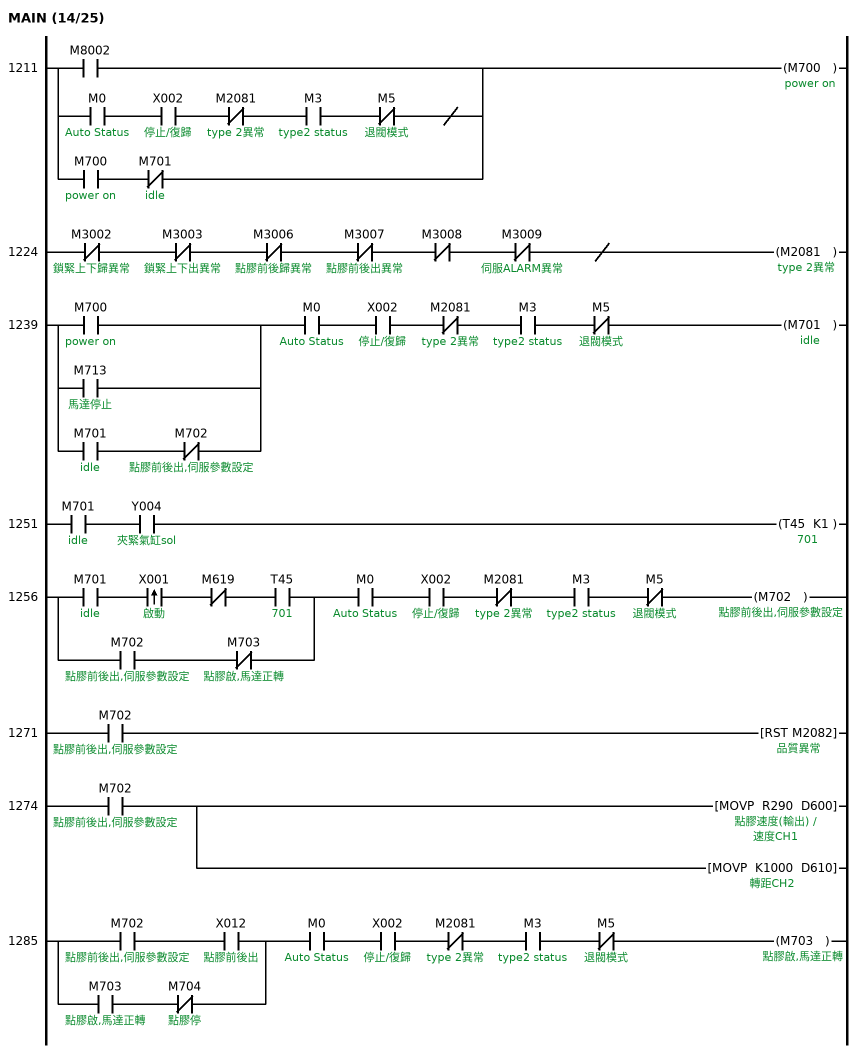
1211  LD      M8002
      LD      M0  ; Auto Status
      AND     X002  ; 停止/復歸
      ANI     M2081  ; type 2異常
      AND     M3  ; type2 status
      ANI     M5  ; 退閥模式
      INV
      ORB
      LD      M700  ; power on
      ANI     M701  ; idle
      ORB
      OUT     M700  ; power on
1224  LDI     M3002  ; 鎖緊上下歸異常
      ANI     M3003  ; 鎖緊上下出異常
      ANI     M3006  ; 點膠前後歸異常
      ANI     M3007  ; 點膠前後出異常
      ANI     M3008
      ANI     M3009  ; 伺服ALARM異常
      INV
      OUT     M2081  ; type 2異常
1239  LD      M700  ; power on
      OR      M713  ; 馬達停止
      LD      M701  ; idle
      ANI     M702  ; 點膠前後出,伺服參數設定
      ORB
      AND     M0  ; Auto Status
      AND     X002  ; 停止/復歸
      ANI     M2081  ; type 2異常
      AND     M3  ; type2 status
      ANI     M5  ; 退閥模式
      OUT     M701  ; idle
1251  LD      M701  ; idle
      AND     Y004  ; 夾緊氣缸sol
      OUT     T45 K1  ; 701
1256  LD      M701  ; idle
      ANDP    X001  ; 啟動
      ANI     M619
      AND     T45  ; 701
      LD      M702  ; 點膠前後出,伺服參數設定
      ANI     M703  ; 點膠啟,馬達正轉
      ORB
      AND     M0  ; Auto Status
      AND     X002  ; 停止/復歸
      ANI     M2081  ; type 2異常
      AND     M3  ; type2 status
      ANI     M5  ; 退閥模式
      OUT     M702  ; 點膠前後出,伺服參數設定
1271  LD      M702  ; 點膠前後出,伺服參數設定
      RST     M2082  ; 品質異常
1274  LD      M702  ; 點膠前後出,伺服參數設定
      MOVP    R290 D600
      MOVP    K1000 D610
1285  LD      M702  ; 點膠前後出,伺服參數設定
      AND     X012  ; 點膠前後出
      LD      M703  ; 點膠啟,馬達正轉
      ANI     M704  ; 點膠停
      ORB
      AND     M0  ; Auto Status
      AND     X002  ; 停止/復歸
      ANI     M2081  ; type 2異常
      AND     M3  ; type2 status
      ANI     M5  ; 退閥模式
      OUT     M703  ; 點膠啟,馬達正轉
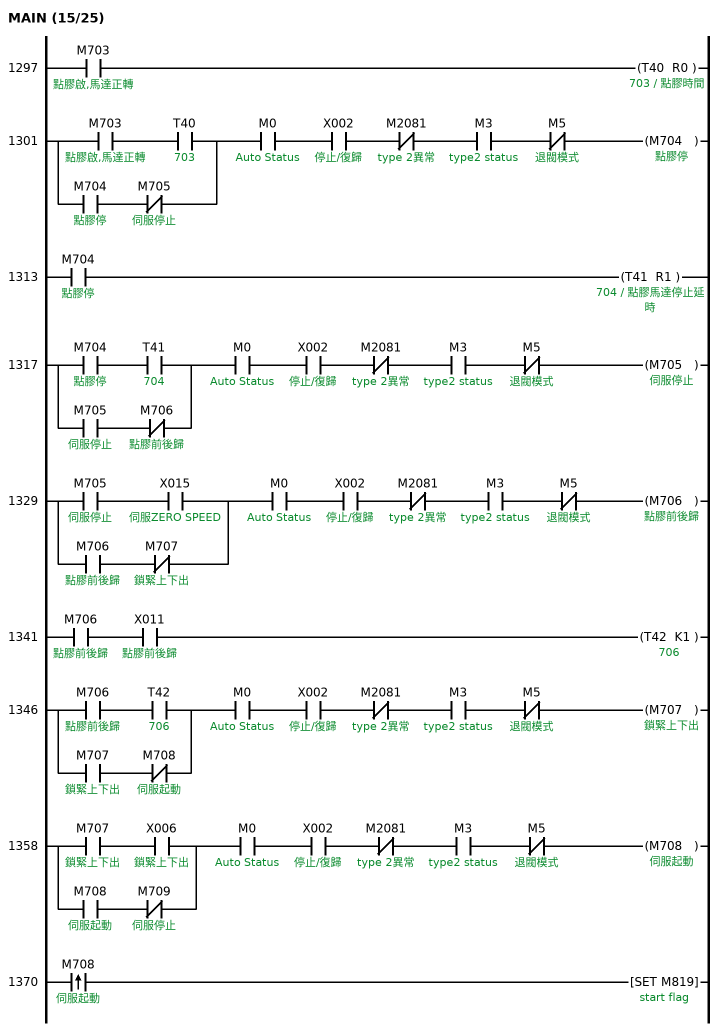
1297  LD      M703  ; 點膠啟,馬達正轉
      OUT     T40 R0  ; 703 / 點膠時間
1301  LD      M703  ; 點膠啟,馬達正轉
      AND     T40  ; 703
      LD      M704  ; 點膠停
      ANI     M705  ; 伺服停止
      ORB
      AND     M0  ; Auto Status
      AND     X002  ; 停止/復歸
      ANI     M2081  ; type 2異常
      AND     M3  ; type2 status
      ANI     M5  ; 退閥模式
      OUT     M704  ; 點膠停
1313  LD      M704  ; 點膠停
      OUT     T41 R1  ; 704 / 點膠馬達停止延時
1317  LD      M704  ; 點膠停
      AND     T41  ; 704
      LD      M705  ; 伺服停止
      ANI     M706  ; 點膠前後歸
      ORB
      AND     M0  ; Auto Status
      AND     X002  ; 停止/復歸
      ANI     M2081  ; type 2異常
      AND     M3  ; type2 status
      ANI     M5  ; 退閥模式
      OUT     M705  ; 伺服停止
1329  LD      M705  ; 伺服停止
      AND     X015  ; 伺服ZERO SPEED
      LD      M706  ; 點膠前後歸
      ANI     M707  ; 鎖緊上下出
      ORB
      AND     M0  ; Auto Status
      AND     X002  ; 停止/復歸
      ANI     M2081  ; type 2異常
      AND     M3  ; type2 status
      ANI     M5  ; 退閥模式
      OUT     M706  ; 點膠前後歸
1341  LD      M706  ; 點膠前後歸
      AND     X011  ; 點膠前後歸
      OUT     T42 K1  ; 706
1346  LD      M706  ; 點膠前後歸
      AND     T42  ; 706
      LD      M707  ; 鎖緊上下出
      ANI     M708  ; 伺服起動
      ORB
      AND     M0  ; Auto Status
      AND     X002  ; 停止/復歸
      ANI     M2081  ; type 2異常
      AND     M3  ; type2 status
      ANI     M5  ; 退閥模式
      OUT     M707  ; 鎖緊上下出
1358  LD      M707  ; 鎖緊上下出
      AND     X006  ; 鎖緊上下出
      LD      M708  ; 伺服起動
      ANI     M709  ; 伺服停止
      ORB
      AND     M0  ; Auto Status
      AND     X002  ; 停止/復歸
      ANI     M2081  ; type 2異常
      AND     M3  ; type2 status
      ANI     M5  ; 退閥模式
      OUT     M708  ; 伺服起動
1370  LDP     M708  ; 伺服起動
      SET     M819  ; start flag
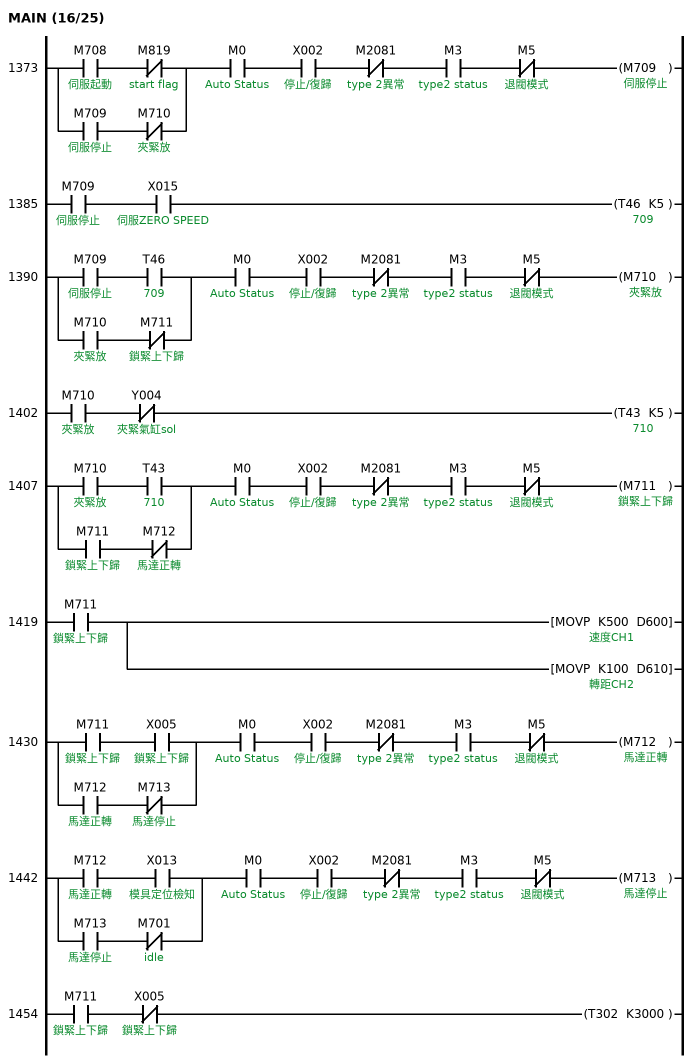
1373  LD      M708  ; 伺服起動
      ANI     M819  ; start flag
      LD      M709  ; 伺服停止
      ANI     M710  ; 夾緊放
      ORB
      AND     M0  ; Auto Status
      AND     X002  ; 停止/復歸
      ANI     M2081  ; type 2異常
      AND     M3  ; type2 status
      ANI     M5  ; 退閥模式
      OUT     M709  ; 伺服停止
1385  LD      M709  ; 伺服停止
      AND     X015  ; 伺服ZERO SPEED
      OUT     T46 K5  ; 709
1390  LD      M709  ; 伺服停止
      AND     T46  ; 709
      LD      M710  ; 夾緊放
      ANI     M711  ; 鎖緊上下歸
      ORB
      AND     M0  ; Auto Status
      AND     X002  ; 停止/復歸
      ANI     M2081  ; type 2異常
      AND     M3  ; type2 status
      ANI     M5  ; 退閥模式
      OUT     M710  ; 夾緊放
1402  LD      M710  ; 夾緊放
      ANI     Y004  ; 夾緊氣缸sol
      OUT     T43 K5  ; 710
1407  LD      M710  ; 夾緊放
      AND     T43  ; 710
      LD      M711  ; 鎖緊上下歸
      ANI     M712  ; 馬達正轉
      ORB
      AND     M0  ; Auto Status
      AND     X002  ; 停止/復歸
      ANI     M2081  ; type 2異常
      AND     M3  ; type2 status
      ANI     M5  ; 退閥模式
      OUT     M711  ; 鎖緊上下歸
1419  LD      M711  ; 鎖緊上下歸
      MOVP    K500 D600
      MOVP    K100 D610
1430  LD      M711  ; 鎖緊上下歸
      AND     X005  ; 鎖緊上下歸
      LD      M712  ; 馬達正轉
      ANI     M713  ; 馬達停止
      ORB
      AND     M0  ; Auto Status
      AND     X002  ; 停止/復歸
      ANI     M2081  ; type 2異常
      AND     M3  ; type2 status
      ANI     M5  ; 退閥模式
      OUT     M712  ; 馬達正轉
1442  LD      M712  ; 馬達正轉
      AND     X013  ; 模具定位檢知
      LD      M713  ; 馬達停止
      ANI     M701  ; idle
      ORB
      AND     M0  ; Auto Status
      AND     X002  ; 停止/復歸
      ANI     M2081  ; type 2異常
      AND     M3  ; type2 status
      ANI     M5  ; 退閥模式
      OUT     M713  ; 馬達停止
1454  LD      M711  ; 鎖緊上下歸
      ANI     X005  ; 鎖緊上下歸
      OUT     T302 K3000
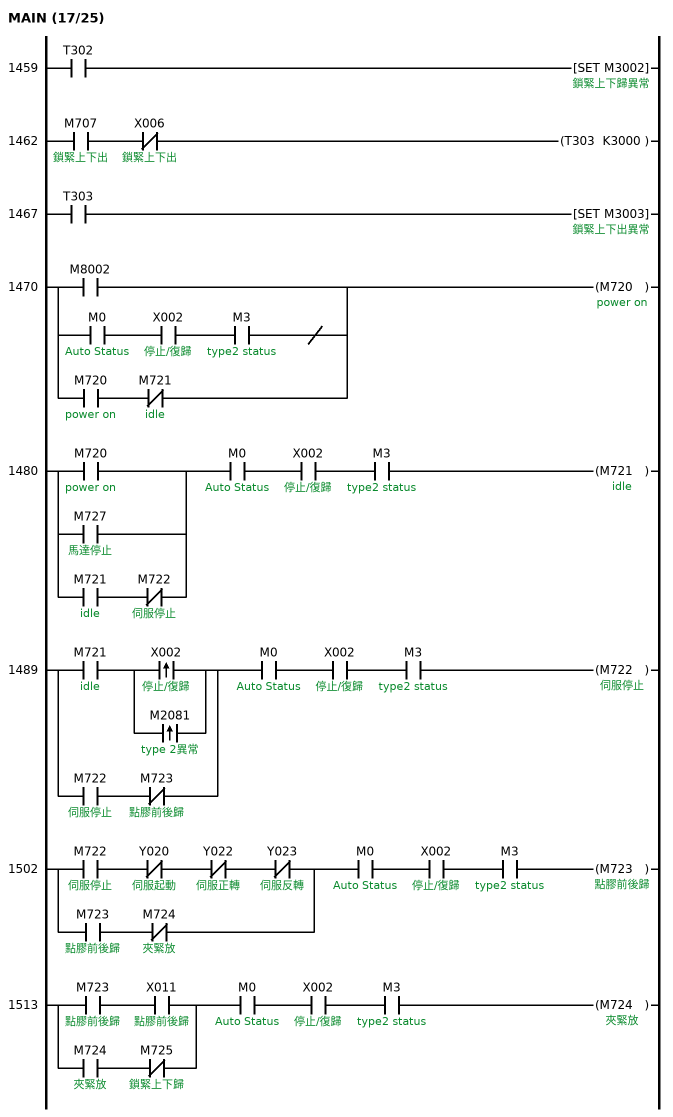
1459  LD      T302
      SET     M3002  ; 鎖緊上下歸異常
1462  LD      M707  ; 鎖緊上下出
      ANI     X006  ; 鎖緊上下出
      OUT     T303 K3000
1467  LD      T303
      SET     M3003  ; 鎖緊上下出異常
1470  LD      M8002
      LD      M0  ; Auto Status
      AND     X002  ; 停止/復歸
      AND     M3  ; type2 status
      INV
      ORB
      LD      M720  ; power on
      ANI     M721  ; idle
      ORB
      OUT     M720  ; power on
1480  LD      M720  ; power on
      OR      M727  ; 馬達停止
      LD      M721  ; idle
      ANI     M722  ; 伺服停止
      ORB
      AND     M0  ; Auto Status
      AND     X002  ; 停止/復歸
      AND     M3  ; type2 status
      OUT     M721  ; idle
1489  LD      M721  ; idle
      LDP     X002  ; 停止/復歸
      ORP     M2081  ; type 2異常
      ANB
      LD      M722  ; 伺服停止
      ANI     M723  ; 點膠前後歸
      ORB
      AND     M0  ; Auto Status
      AND     X002  ; 停止/復歸
      AND     M3  ; type2 status
      OUT     M722  ; 伺服停止
1502  LD      M722  ; 伺服停止
      ANI     Y020  ; 伺服起動
      ANI     Y022  ; 伺服正轉
      ANI     Y023  ; 伺服反轉
      LD      M723  ; 點膠前後歸
      ANI     M724  ; 夾緊放
      ORB
      AND     M0  ; Auto Status
      AND     X002  ; 停止/復歸
      AND     M3  ; type2 status
      OUT     M723  ; 點膠前後歸
1513  LD      M723  ; 點膠前後歸
      AND     X011  ; 點膠前後歸
      LD      M724  ; 夾緊放
      ANI     M725  ; 鎖緊上下歸
      ORB
      AND     M0  ; Auto Status
      AND     X002  ; 停止/復歸
      AND     M3  ; type2 status
      OUT     M724  ; 夾緊放
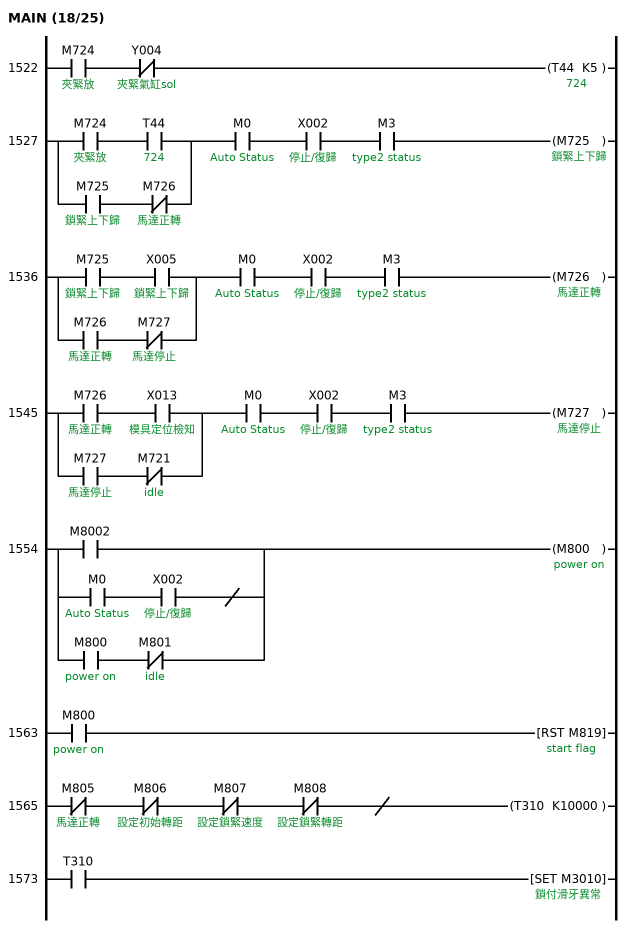
1522  LD      M724  ; 夾緊放
      ANI     Y004  ; 夾緊氣缸sol
      OUT     T44 K5  ; 724
1527  LD      M724  ; 夾緊放
      AND     T44  ; 724
      LD      M725  ; 鎖緊上下歸
      ANI     M726  ; 馬達正轉
      ORB
      AND     M0  ; Auto Status
      AND     X002  ; 停止/復歸
      AND     M3  ; type2 status
      OUT     M725  ; 鎖緊上下歸
1536  LD      M725  ; 鎖緊上下歸
      AND     X005  ; 鎖緊上下歸
      LD      M726  ; 馬達正轉
      ANI     M727  ; 馬達停止
      ORB
      AND     M0  ; Auto Status
      AND     X002  ; 停止/復歸
      AND     M3  ; type2 status
      OUT     M726  ; 馬達正轉
1545  LD      M726  ; 馬達正轉
      AND     X013  ; 模具定位檢知
      LD      M727  ; 馬達停止
      ANI     M721  ; idle
      ORB
      AND     M0  ; Auto Status
      AND     X002  ; 停止/復歸
      AND     M3  ; type2 status
      OUT     M727  ; 馬達停止
1554  LD      M8002
      LD      M0  ; Auto Status
      AND     X002  ; 停止/復歸
      INV
      ORB
      LD      M800  ; power on
      ANI     M801  ; idle
      ORB
      OUT     M800  ; power on
1563  LD      M800  ; power on
      RST     M819  ; start flag
1565  LDI     M805  ; 馬達正轉
      ANI     M806  ; 設定初始轉距
      ANI     M807  ; 設定鎖緊速度
      ANI     M808  ; 設定鎖緊轉距
      INV
      OUT     T310 K10000
1573  LD      T310
      SET     M3010  ; 鎖付滑牙異常
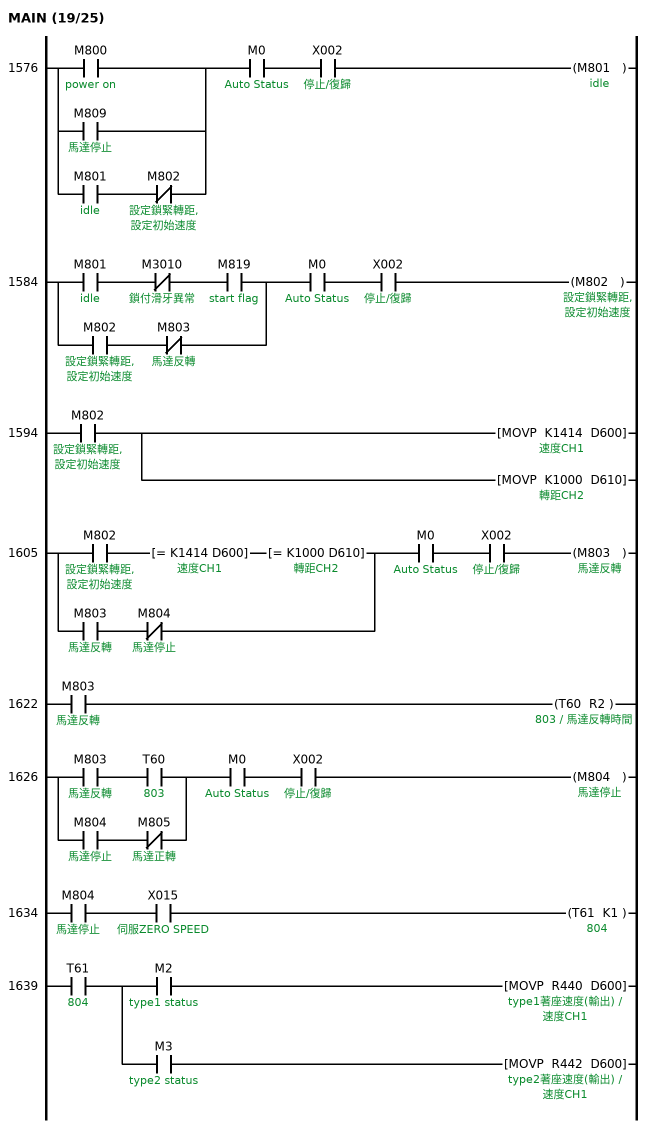
1576  LD      M800  ; power on
      OR      M809  ; 馬達停止
      LD      M801  ; idle
      ANI     M802  ; 設定鎖緊轉距,設定初始速度
      ORB
      AND     M0  ; Auto Status
      AND     X002  ; 停止/復歸
      OUT     M801  ; idle
1584  LD      M801  ; idle
      ANI     M3010  ; 鎖付滑牙異常
      AND     M819  ; start flag
      LD      M802  ; 設定鎖緊轉距,設定初始速度
      ANI     M803  ; 馬達反轉
      ORB
      AND     M0  ; Auto Status
      AND     X002  ; 停止/復歸
      OUT     M802  ; 設定鎖緊轉距,設定初始速度
1594  LD      M802  ; 設定鎖緊轉距,設定初始速度
      MOVP    K1414 D600
      MOVP    K1000 D610
1605  LD      M802  ; 設定鎖緊轉距,設定初始速度
      AND=    K1414 D600  ; 速度CH1
      AND=    K1000 D610  ; 轉距CH2
      LD      M803  ; 馬達反轉
      ANI     M804  ; 馬達停止
      ORB
      AND     M0  ; Auto Status
      AND     X002  ; 停止/復歸
      OUT     M803  ; 馬達反轉
1622  LD      M803  ; 馬達反轉
      OUT     T60 R2  ; 803 / 馬達反轉時間
1626  LD      M803  ; 馬達反轉
      AND     T60  ; 803
      LD      M804  ; 馬達停止
      ANI     M805  ; 馬達正轉
      ORB
      AND     M0  ; Auto Status
      AND     X002  ; 停止/復歸
      OUT     M804  ; 馬達停止
1634  LD      M804  ; 馬達停止
      AND     X015  ; 伺服ZERO SPEED
      OUT     T61 K1  ; 804
1639  LD      T61  ; 804
      MPS
      AND     M2  ; type1 status
      MOVP    R440 D600  ; type1著座速度(輸出)
      MPP
      AND     M3  ; type2 status
      MOVP    R442 D600  ; type2著座速度(輸出)
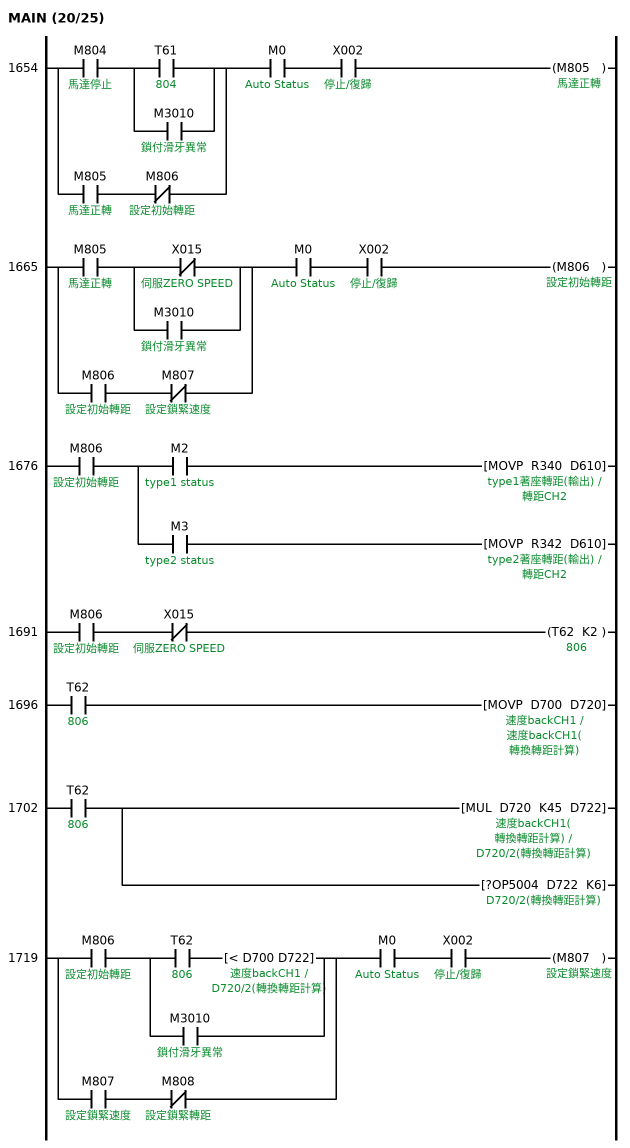
1654  LD      M804  ; 馬達停止
      LD      T61  ; 804
      OR      M3010  ; 鎖付滑牙異常
      ANB
      LD      M805  ; 馬達正轉
      ANI     M806  ; 設定初始轉距
      ORB
      AND     M0  ; Auto Status
      AND     X002  ; 停止/復歸
      OUT     M805  ; 馬達正轉
1665  LD      M805  ; 馬達正轉
      LDI     X015  ; 伺服ZERO SPEED
      OR      M3010  ; 鎖付滑牙異常
      ANB
      LD      M806  ; 設定初始轉距
      ANI     M807  ; 設定鎖緊速度
      ORB
      AND     M0  ; Auto Status
      AND     X002  ; 停止/復歸
      OUT     M806  ; 設定初始轉距
1676  LD      M806  ; 設定初始轉距
      MPS
      AND     M2  ; type1 status
      MOVP    R340 D610  ; type1著座轉距(輸出)
      MPP
      AND     M3  ; type2 status
      MOVP    R342 D610  ; type2著座轉距(輸出)
1691  LD      M806  ; 設定初始轉距
      ANI     X015  ; 伺服ZERO SPEED
      OUT     T62 K2  ; 806
1696  LD      T62  ; 806
      MOVP    D700 D720  ; 速度backCH1(轉換轉距計算)
1702  LD      T62  ; 806
      MUL     D720 K45 D722  ; D720/2(轉換轉距計算)
      ?OP5004 D722 K6
1719  LD      M806  ; 設定初始轉距
      LD      T62  ; 806
      AND<    D700 D722  ; 速度backCH1 / D720/2(轉換轉距計算)
      OR      M3010  ; 鎖付滑牙異常
      ANB
      LD      M807  ; 設定鎖緊速度
      ANI     M808  ; 設定鎖緊轉距
      ORB
      AND     M0  ; Auto Status
      AND     X002  ; 停止/復歸
      OUT     M807  ; 設定鎖緊速度
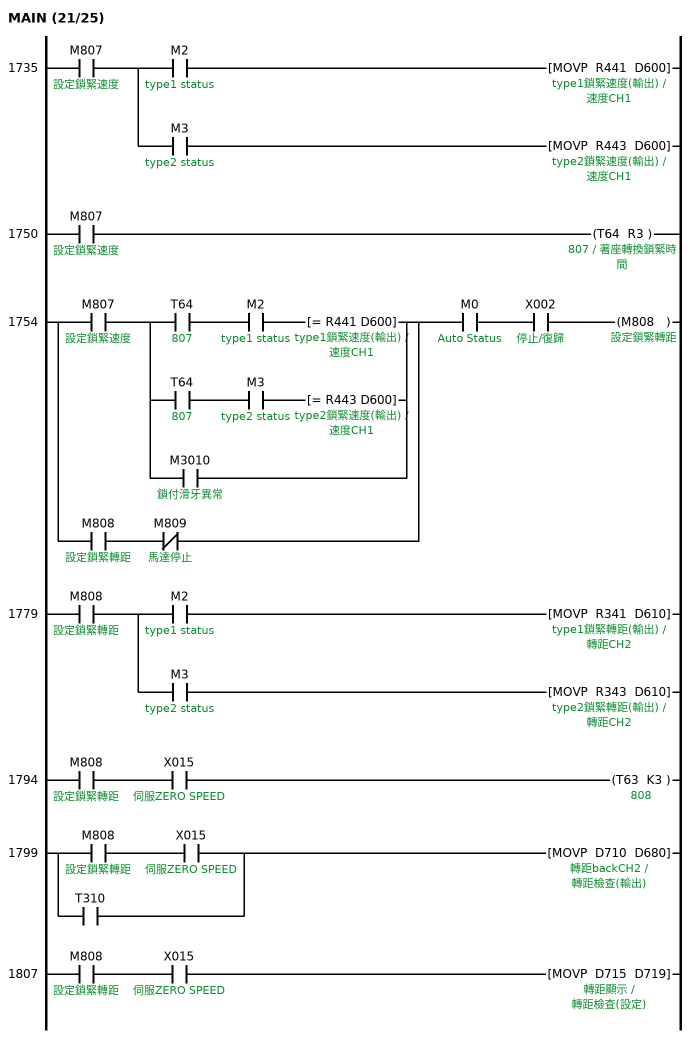
1735  LD      M807  ; 設定鎖緊速度
      MPS
      AND     M2  ; type1 status
      MOVP    R441 D600  ; type1鎖緊速度(輸出)
      MPP
      AND     M3  ; type2 status
      MOVP    R443 D600  ; type2鎖緊速度(輸出)
1750  LD      M807  ; 設定鎖緊速度
      OUT     T64 R3  ; 807 / 著座轉換鎖緊時間
1754  LD      M807  ; 設定鎖緊速度
      LD      T64  ; 807
      AND     M2  ; type1 status
      AND=    R441 D600  ; type1鎖緊速度(輸出) / 速度CH1
      LD      T64  ; 807
      AND     M3  ; type2 status
      AND=    R443 D600  ; type2鎖緊速度(輸出) / 速度CH1
      ORB
      OR      M3010  ; 鎖付滑牙異常
      ANB
      LD      M808  ; 設定鎖緊轉距
      ANI     M809  ; 馬達停止
      ORB
      AND     M0  ; Auto Status
      AND     X002  ; 停止/復歸
      OUT     M808  ; 設定鎖緊轉距
1779  LD      M808  ; 設定鎖緊轉距
      MPS
      AND     M2  ; type1 status
      MOVP    R341 D610  ; type1鎖緊轉距(輸出)
      MPP
      AND     M3  ; type2 status
      MOVP    R343 D610  ; type2鎖緊轉距(輸出)
1794  LD      M808  ; 設定鎖緊轉距
      AND     X015  ; 伺服ZERO SPEED
      OUT     T63 K3  ; 808
1799  LD      M808  ; 設定鎖緊轉距
      AND     X015  ; 伺服ZERO SPEED
      OR      T310
      MOVP    D710 D680  ; 轉距檢查(輸出)
1807  LD      M808  ; 設定鎖緊轉距
      AND     X015  ; 伺服ZERO SPEED
      MOVP    D715 D719  ; 轉距顯示 / 轉距檢查(設定)
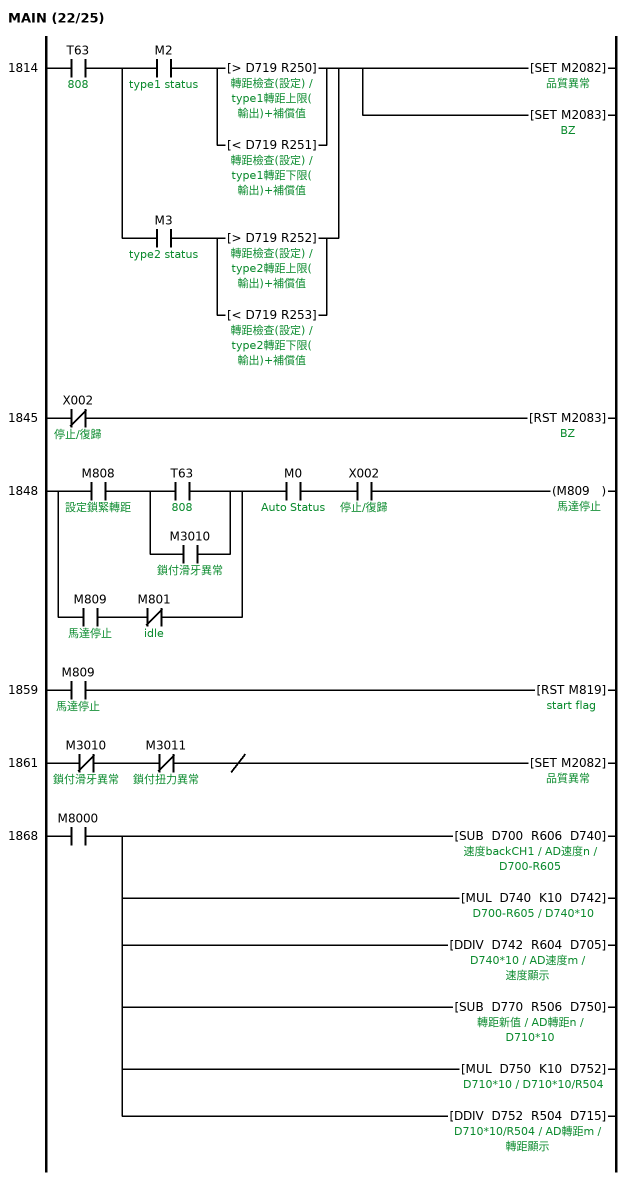
1814  LD      T63  ; 808
      LD      M2  ; type1 status
      LD>     D719 R250  ; 轉距檢查(設定) / type1轉距上限(輸出)+補償值
      OR<     D719 R251  ; 轉距檢查(設定) / type1轉距下限(輸出)+補償值
      ANB
      LD      M3  ; type2 status
      LD>     D719 R252  ; 轉距檢查(設定) / type2轉距上限(輸出)+補償值
      OR<     D719 R253  ; 轉距檢查(設定) / type2轉距下限(輸出)+補償值
      ANB
      ORB
      ANB
      SET     M2082  ; 品質異常
      SET     M2083  ; BZ
1845  LDI     X002  ; 停止/復歸
      RST     M2083  ; BZ
1848  LD      M808  ; 設定鎖緊轉距
      LD      T63  ; 808
      OR      M3010  ; 鎖付滑牙異常
      ANB
      LD      M809  ; 馬達停止
      ANI     M801  ; idle
      ORB
      AND     M0  ; Auto Status
      AND     X002  ; 停止/復歸
      OUT     M809  ; 馬達停止
1859  LD      M809  ; 馬達停止
      RST     M819  ; start flag
1861  LDI     M3010  ; 鎖付滑牙異常
      ANI     M3011  ; 鎖付扭力異常
      INV
      SET     M2082  ; 品質異常
1868  LD      M8000
      SUB     D700 R606 D740  ; AD速度n / D700-R605
      MUL     D740 K10 D742  ; D740*10
      DDIV    D742 R604 D705  ; AD速度m / 速度顯示
      SUB     D770 R506 D750  ; AD轉距n / D710*10
      MUL     D750 K10 D752  ; D710*10/R504
      DDIV    D752 R504 D715  ; AD轉距m
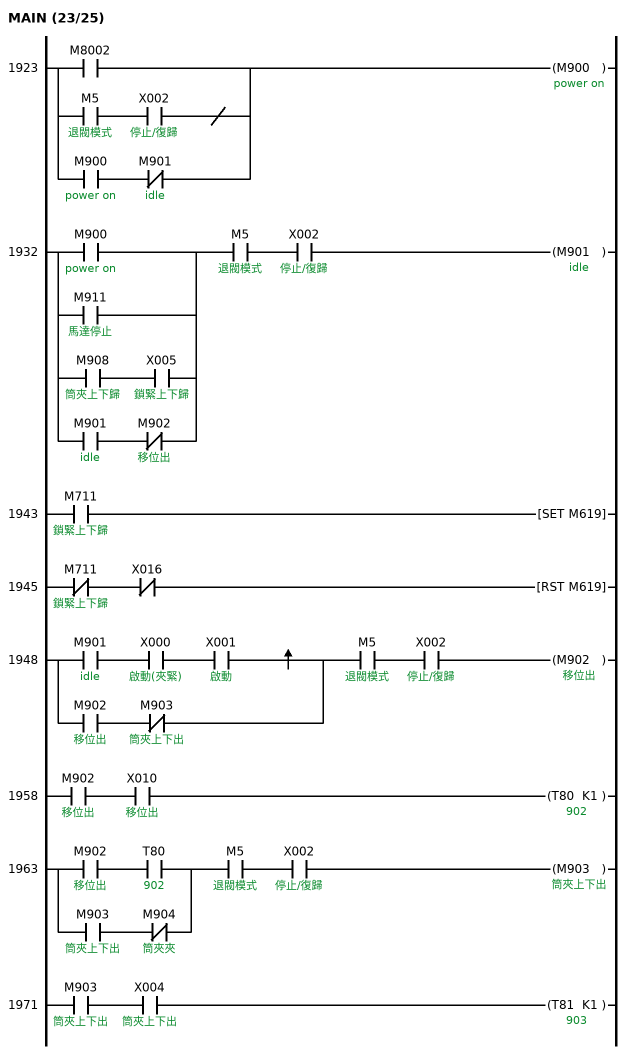
1923  LD      M8002
      LD      M5  ; 退閥模式
      AND     X002  ; 停止/復歸
      INV
      ORB
      LD      M900  ; power on
      ANI     M901  ; idle
      ORB
      OUT     M900  ; power on
1932  LD      M900  ; power on
      OR      M911  ; 馬達停止
      LD      M908  ; 筒夾上下歸
      AND     X005  ; 鎖緊上下歸
      ORB
      LD      M901  ; idle
      ANI     M902  ; 移位出
      ORB
      AND     M5  ; 退閥模式
      AND     X002  ; 停止/復歸
      OUT     M901  ; idle
1943  LD      M711  ; 鎖緊上下歸
      SET     M619
1945  LDI     M711  ; 鎖緊上下歸
      ANI     X016
      RST     M619
1948  LD      M901  ; idle
      AND     X000  ; 啟動(夾緊)
      AND     X001  ; 啟動
      MEP
      LD      M902  ; 移位出
      ANI     M903  ; 筒夾上下出
      ORB
      AND     M5  ; 退閥模式
      AND     X002  ; 停止/復歸
      OUT     M902  ; 移位出
1958  LD      M902  ; 移位出
      AND     X010  ; 移位出
      OUT     T80 K1  ; 902
1963  LD      M902  ; 移位出
      AND     T80  ; 902
      LD      M903  ; 筒夾上下出
      ANI     M904  ; 筒夾夾
      ORB
      AND     M5  ; 退閥模式
      AND     X002  ; 停止/復歸
      OUT     M903  ; 筒夾上下出
1971  LD      M903  ; 筒夾上下出
      AND     X004  ; 筒夾上下出
      OUT     T81 K1  ; 903
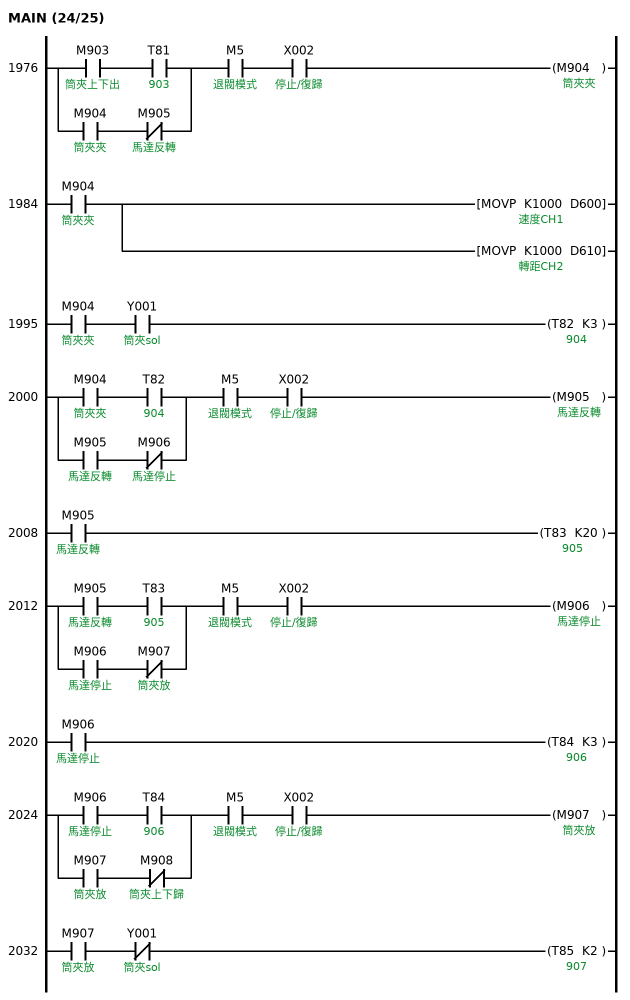
1976  LD      M903  ; 筒夾上下出
      AND     T81  ; 903
      LD      M904  ; 筒夾夾
      ANI     M905  ; 馬達反轉
      ORB
      AND     M5  ; 退閥模式
      AND     X002  ; 停止/復歸
      OUT     M904  ; 筒夾夾
1984  LD      M904  ; 筒夾夾
      MOVP    K1000 D600
      MOVP    K1000 D610
1995  LD      M904  ; 筒夾夾
      AND     Y001  ; 筒夾sol
      OUT     T82 K3  ; 904
2000  LD      M904  ; 筒夾夾
      AND     T82  ; 904
      LD      M905  ; 馬達反轉
      ANI     M906  ; 馬達停止
      ORB
      AND     M5  ; 退閥模式
      AND     X002  ; 停止/復歸
      OUT     M905  ; 馬達反轉
2008  LD      M905  ; 馬達反轉
      OUT     T83 K20  ; 905
2012  LD      M905  ; 馬達反轉
      AND     T83  ; 905
      LD      M906  ; 馬達停止
      ANI     M907  ; 筒夾放
      ORB
      AND     M5  ; 退閥模式
      AND     X002  ; 停止/復歸
      OUT     M906  ; 馬達停止
2020  LD      M906  ; 馬達停止
      OUT     T84 K3  ; 906
2024  LD      M906  ; 馬達停止
      AND     T84  ; 906
      LD      M907  ; 筒夾放
      ANI     M908  ; 筒夾上下歸
      ORB
      AND     M5  ; 退閥模式
      AND     X002  ; 停止/復歸
      OUT     M907  ; 筒夾放
2032  LD      M907  ; 筒夾放
      ANI     Y001  ; 筒夾sol
      OUT     T85 K2  ; 907
